        GetEndpointFromOrchestrationForm.endpoint TO F_EQ.IN2;
        F_EQ.OUT TO NoServiceAvailable.check;
        E_SR.Q TO SERVER_1.QI;
        Service1.arrowheadService TO RegisterService2.providedService;
        FieldsToArrowheadSystem.arrowheadSystem TO RegisterService2.provider;
        GET_STRUCT_VALUE1.OUT TO GetEndpointFromOrchestrationForm.orchestrationForm;
        FieldsToServiceRequestForm.serviceRequestForm TO RequestOrchestrationForm.serviceRequestForm;
        RequestOrchestrationForm.orchestrationResponse TO GET_STRUCT_VALUE1.IN_ARRAY;
      END_CONNECTIONS
      ADAPTER_CONNECTIONS
        RequestOrchestrationForm.requestOrchestration TO RequestOrchestrationHTTP.requestOrchestration;
      END_CONNECTIONS
    END_RESOURCE
    RESOURCE OrchestrationWithRules : EMB_RES
      FBS
        FieldsToArrowheadSystem : FieldsToArrowheadSystem(systemName := %systemName%, address := %testAddress%, port := %systemPort%);
        Service1 : FieldsToArrowheadService(serviceDefinition := %serviceDefinition%, interfaces := ["JSON", "XML"], serviceMetadata := %serviceMetadata%);
        F_EQ : F_EQ(IN1 := %emptyEndpoint%);
        NoServiceAvailable : TEST_CONDITION;
        SERVER_1 : SERVER_1(ID := http[/serviceTest/start]);
        E_SR : E_SR;
        SUBL_0 : SUBL_0(ID := %test7Ended%);
        PUBL_0 : PUBL_0(ID := %test8Ended%);
        F_EQ_1 : F_EQ(IN1 := %validEndpoint%);
        ServiceAvailable : TEST_CONDITION;
        E_SR_1 : E_SR;
        E_SWITCH : E_SWITCH;
        CLIENT_1_2 : CLIENT_1_2(QI := 1, ID := http[%authRuleEndpoint%; POST; application/json]], SD_1 := STRING#%authRuleData%);
        CLIENT_1_2_1 : CLIENT_1_2(QI := 1, ID := http[%orchStoreEndpoint%; POST; application/json]], SD_1 := STRING#%orchRuleData%);
        STRING2STRING : STRING2STRING;
      END_FBS
      SUBAPPS
        RegisterService2 : RegisterServicePartialHTTP(serviceURI := %serviceURI%, version := %serviceVersion%, udp := false, metadata := %metadata%, SRendpoint := %serviceRegistryAddress%);
        GetEndpointFromOrchestrationHTTPPFull : GetEndpointFromOrchestrationHTTPPFull(systemName := %systemName%, address := %testAddress%, port := %systemPort%, serviceDefinition := %serviceDefinition%, interfaces := ["JSON", "XML"], serviceMetadata := %serviceMetadata%, orchestratorEndpoint := %orchestratorAddress%, INDEX := 0);
      END_SUBAPPS
      SUBAPPLICATION Sequencer_1
        EVENT_INPUT
          Next;
        END_EVENT
        EVENT_OUTPUT
          E0;
          E1;
          E2;
          E3;
          E4;
          E5;
          E6;
          E7;
          E8;
          E9;
          E10;
          E11;
          E12;
          E13;
          E14;
          E15;
        END_EVENT
      END_SUBAPPLICATION
      EVENT_CONNECTIONS
        FieldsToArrowheadSystem.CNF TO Service1.REQ;
        F_EQ.CNF TO NoServiceAvailable.REQ;
        E_SR.EO TO SERVER_1.INIT;
        SUBL_0.IND TO FieldsToArrowheadSystem.REQ;
        RegisterService2.doneUnregister TO Sequencer_1.Next;
        RegisterService2.doneRegister TO Sequencer_1.Next;
        NoServiceAvailable.CNF TO Sequencer_1.Next;
        F_EQ_1.CNF TO ServiceAvailable.REQ;
        E_SWITCH.EO0 TO F_EQ.REQ;
        E_SWITCH.EO1 TO F_EQ_1.REQ;
        Sequencer_1.E2 TO RegisterService2.register;
        E_SR_1.EO TO Sequencer_1.Next;
        START.WARM TO SUBL_0.INIT;
        SERVER_1.INITO TO Sequencer_1.Next;
        CLIENT_1_2.INITO TO CLIENT_1_2.REQ;
        CLIENT_1_2.CNF TO CLIENT_1_2_1.INIT;
        CLIENT_1_2_1.INITO TO CLIENT_1_2_1.REQ;
        Sequencer_1.E0 TO CLIENT_1_2.INIT;
        SERVER_1.IND TO STRING2STRING.REQ;
        STRING2STRING.CNF TO SERVER_1.RSP;
        Sequencer_1.E3 TO E_SR_1.S;
        Sequencer_1.E5 TO E_SR.S;
        Sequencer_1.E7 TO RegisterService2.unregister;
        Sequencer_1.E8 TO E_SR_1.R;
        Sequencer_1.E10 TO E_SR.R;
        START.COLD TO SUBL_0.INIT;
        Service1.CNF TO Sequencer_1.Next;
        Sequencer_1.E11 TO GetEndpointFromOrchestrationHTTPPFull.REQ;
        Sequencer_1.E9 TO GetEndpointFromOrchestrationHTTPPFull.REQ;
        Sequencer_1.E6 TO GetEndpointFromOrchestrationHTTPPFull.REQ;
        Sequencer_1.E4 TO GetEndpointFromOrchestrationHTTPPFull.REQ;
        Sequencer_1.E1 TO GetEndpointFromOrchestrationHTTPPFull.REQ;
        GetEndpointFromOrchestrationHTTPPFull.CNF TO E_SWITCH.EI;
        CLIENT_1_2_1.CNF TO Sequencer_1.Next;
        ServiceAvailable.CNF TO Sequencer_1.Next;
        SUBL_0.INITO TO PUBL_0.INIT;
        Sequencer_1.E12 TO PUBL_0.REQ;
      END_CONNECTIONS
      DATA_CONNECTIONS
        F_EQ.OUT TO NoServiceAvailable.check;
        E_SR.Q TO SERVER_1.QI;
        Service1.arrowheadService TO RegisterService2.providedService;
        FieldsToArrowheadSystem.arrowheadSystem TO RegisterService2.provider;
        F_EQ_1.OUT TO ServiceAvailable.check;
        E_SR_1.Q TO E_SWITCH.G;
        SERVER_1.RD_1 TO STRING2STRING.IN;
        STRING2STRING.OUT TO SERVER_1.SD_1;
        GetEndpointFromOrchestrationHTTPPFull.endpoint TO F_EQ_1.IN2;
        GetEndpointFromOrchestrationHTTPPFull.endpoint TO F_EQ.IN2;
      END_CONNECTIONS
    END_RESOURCE
    RESOURCE PublishSubscribe : EMB_RES
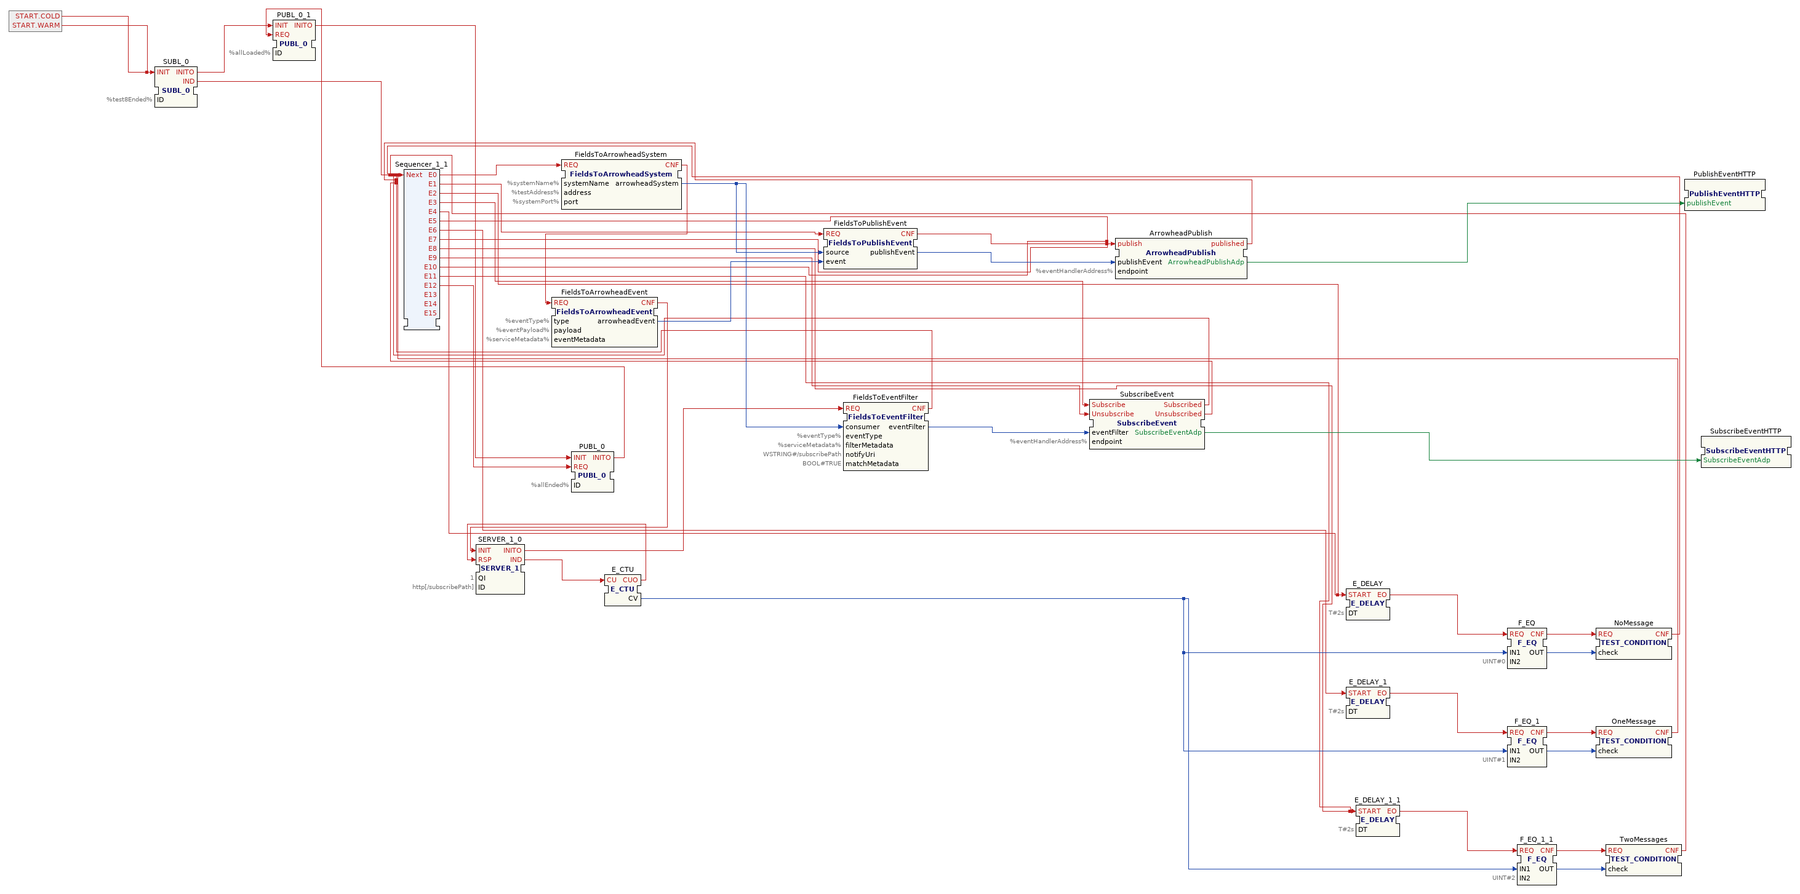
      FBS
        FieldsToArrowheadSystem : FieldsToArrowheadSystem(systemName := %systemName%, address := %testAddress%, port := %systemPort%);
        FieldsToPublishEvent : FieldsToPublishEvent;
        ArrowheadPublish : ArrowheadPublish(endpoint := %eventHandlerAddress%);
        FieldsToArrowheadEvent : FieldsToArrowheadEvent(type := %eventType%, payload := %eventPayload%, eventMetadata := %serviceMetadata%);
        SubscribeEvent : SubscribeEvent(endpoint := %eventHandlerAddress%);
        FieldsToEventFilter : FieldsToEventFilter(eventType := %eventType%, filterMetadata := %serviceMetadata%, notifyUri := WSTRING#/subscribePath, matchMetadata := BOOL#TRUE);
        E_CTU : E_CTU;
        F_EQ : F_EQ(IN2 := UINT#0);
        E_DELAY : E_DELAY(DT := T#2s);
        NoMessage : TEST_CONDITION;
        E_DELAY_1 : E_DELAY(DT := T#2s);
        F_EQ_1 : F_EQ(IN2 := UINT#1);
        OneMessage : TEST_CONDITION;
        E_DELAY_1_1 : E_DELAY(DT := T#2s);
        TwoMessages : TEST_CONDITION;
        F_EQ_1_1 : F_EQ(IN2 := UINT#2);
        SERVER_1_0 : SERVER_1(QI := 1, ID := http[/subscribePath]);
        PUBL_0_1 : PUBL_0(ID := %allLoaded%);
        SUBL_0 : SUBL_0(ID := %test8Ended%);
        PUBL_0 : PUBL_0(ID := %allEnded%);
        PublishEventHTTP : PublishEventHTTP;
        SubscribeEventHTTP : SubscribeEventHTTP;
      END_FBS
      SUBAPPLICATION Sequencer_1_1
        EVENT_INPUT
          Next;
        END_EVENT
        EVENT_OUTPUT
          E0;
          E1;
          E2;
          E3;
          E4;
          E5;
          E6;
          E7;
          E8;
          E9;
          E10;
          E11;
          E12;
          E13;
          E14;
          E15;
        END_EVENT
      END_SUBAPPLICATION
      EVENT_CONNECTIONS
        FieldsToPublishEvent.CNF TO ArrowheadPublish.publish;
        FieldsToArrowheadSystem.CNF TO FieldsToArrowheadEvent.REQ;
        E_DELAY.EO TO F_EQ.REQ;
        F_EQ.CNF TO NoMessage.REQ;
        E_DELAY_1.EO TO F_EQ_1.REQ;
        F_EQ_1.CNF TO OneMessage.REQ;
        E_DELAY_1_1.EO TO F_EQ_1_1.REQ;
        F_EQ_1_1.CNF TO TwoMessages.REQ;
        TwoMessages.CNF TO Sequencer_1_1.Next;
        OneMessage.CNF TO Sequencer_1_1.Next;
        NoMessage.CNF TO Sequencer_1_1.Next;
        FieldsToEventFilter.CNF TO Sequencer_1_1.Next;
        Sequencer_1_1.E0 TO FieldsToArrowheadSystem.REQ;
        Sequencer_1_1.E1 TO FieldsToPublishEvent.REQ;
        Sequencer_1_1.E2 TO E_DELAY.START;
        Sequencer_1_1.E3 TO SubscribeEvent.Subscribe;
        Sequencer_1_1.E4 TO E_DELAY.START;
        Sequencer_1_1.E5 TO ArrowheadPublish.publish;
        Sequencer_1_1.E6 TO E_DELAY_1.START;
        Sequencer_1_1.E7 TO ArrowheadPublish.publish;
        Sequencer_1_1.E8 TO E_DELAY_1_1.START;
        Sequencer_1_1.E9 TO SubscribeEvent.Unsubscribe;
        Sequencer_1_1.E10 TO ArrowheadPublish.publish;
        Sequencer_1_1.E11 TO E_DELAY_1_1.START;
        ArrowheadPublish.published TO Sequencer_1_1.Next;
        SubscribeEvent.Subscribed TO Sequencer_1_1.Next;
        FieldsToArrowheadEvent.CNF TO SERVER_1_0.INIT;
        E_CTU.CUO TO SERVER_1_0.RSP;
        SERVER_1_0.INITO TO FieldsToEventFilter.REQ;
        SERVER_1_0.IND TO E_CTU.CU;
        SubscribeEvent.Unsubscribed TO Sequencer_1_1.Next;
        SUBL_0.INITO TO PUBL_0_1.INIT;
        START.COLD TO SUBL_0.INIT;
        START.WARM TO SUBL_0.INIT;
        SUBL_0.IND TO Sequencer_1_1.Next;
        PUBL_0_1.INITO TO PUBL_0.INIT;
        PUBL_0.INITO TO PUBL_0_1.REQ;
        Sequencer_1_1.E12 TO PUBL_0.REQ;
      END_CONNECTIONS
      DATA_CONNECTIONS
        FieldsToArrowheadSystem.arrowheadSystem TO FieldsToPublishEvent.source;
        FieldsToPublishEvent.publishEvent TO ArrowheadPublish.publishEvent;
        FieldsToArrowheadEvent.arrowheadEvent TO FieldsToPublishEvent.event;
        FieldsToArrowheadSystem.arrowheadSystem TO FieldsToEventFilter.consumer;
        FieldsToEventFilter.eventFilter TO SubscribeEvent.eventFilter;
        E_CTU.CV TO F_EQ.IN1;
        F_EQ.OUT TO NoMessage.check;
        E_CTU.CV TO F_EQ_1.IN1;
        F_EQ_1.OUT TO OneMessage.check;
        F_EQ_1_1.OUT TO TwoMessages.check;
        E_CTU.CV TO F_EQ_1_1.IN1;
      END_CONNECTIONS
      ADAPTER_CONNECTIONS
        ArrowheadPublish.ArrowheadPublishAdp TO PublishEventHTTP.publishEvent;
        SubscribeEvent.SubscribeEventAdp TO SubscribeEventHTTP.SubscribeEventAdp;
      END_CONNECTIONS
    END_RESOURCE
  END_DEVICE
  DEVICE OpcUaTest : FORTE_PC(MGR_ID := %opcuaTestAddress%)
    {SET_ATTRIBUTE(Profile, HOLOBLOC)} (* device profile *)
    RESOURCE cleanAll : EMB_RES
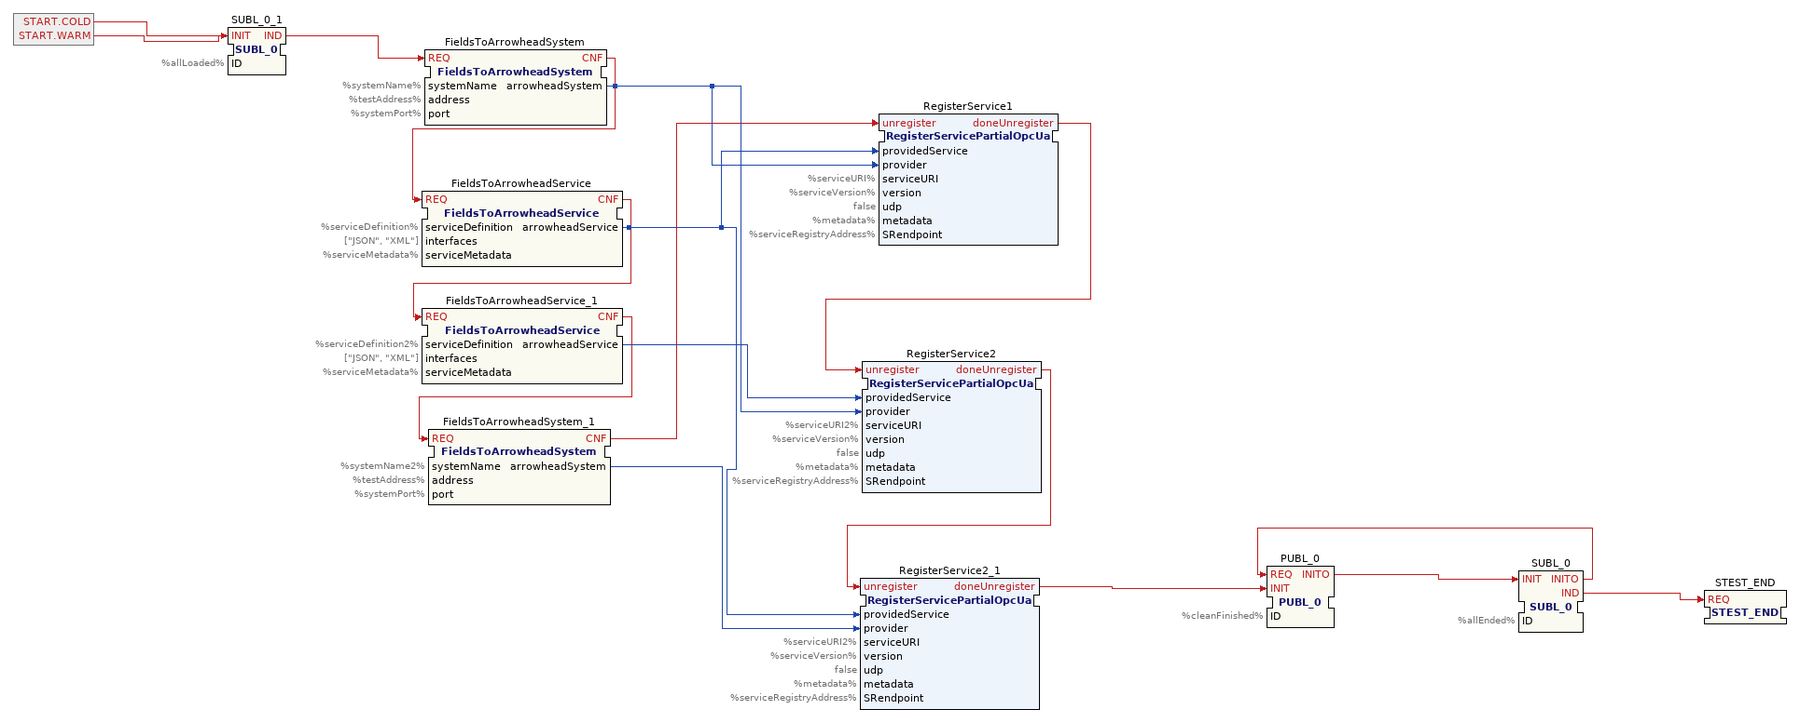
      FBS
        PUBL_0 : PUBL_0(ID := %cleanFinished%);
        FieldsToArrowheadSystem : FieldsToArrowheadSystem(systemName := %systemName%, address := %testAddress%, port := %systemPort%);
        FieldsToArrowheadService : FieldsToArrowheadService(serviceDefinition := %serviceDefinition%, interfaces := ["JSON", "XML"], serviceMetadata := %serviceMetadata%);
        FieldsToArrowheadService_1 : FieldsToArrowheadService(serviceDefinition := %serviceDefinition2%, interfaces := ["JSON", "XML"], serviceMetadata := %serviceMetadata%);
        FieldsToArrowheadSystem_1 : FieldsToArrowheadSystem(systemName := %systemName2%, address := %testAddress%, port := %systemPort%);
        SUBL_0 : SUBL_0(ID := %allEnded%);
        STEST_END : STEST_END;
        SUBL_0_1 : SUBL_0(ID := %allLoaded%);
      END_FBS
      SUBAPPS
        RegisterService1 : RegisterServicePartialOpcUa(serviceURI := %serviceURI%, version := %serviceVersion%, udp := false, metadata := %metadata%, SRendpoint := %serviceRegistryAddress%);
        RegisterService2_1 : RegisterServicePartialOpcUa(serviceURI := %serviceURI2%, version := %serviceVersion%, udp := false, metadata := %metadata%, SRendpoint := %serviceRegistryAddress%);
        RegisterService2 : RegisterServicePartialOpcUa(serviceURI := %serviceURI2%, version := %serviceVersion%, udp := false, metadata := %metadata%, SRendpoint := %serviceRegistryAddress%);
      END_SUBAPPS
      EVENT_CONNECTIONS
        FieldsToArrowheadSystem.CNF TO FieldsToArrowheadService.REQ;
        FieldsToArrowheadService.CNF TO FieldsToArrowheadService_1.REQ;
        FieldsToArrowheadService_1.CNF TO FieldsToArrowheadSystem_1.REQ;
        PUBL_0.INITO TO SUBL_0.INIT;
        SUBL_0.INITO TO PUBL_0.REQ;
        SUBL_0.IND TO STEST_END.REQ;
        START.COLD TO SUBL_0_1.INIT;
        START.WARM TO SUBL_0_1.INIT;
        FieldsToArrowheadSystem_1.CNF TO RegisterService1.unregister;
        RegisterService2_1.doneUnregister TO PUBL_0.INIT;
        RegisterService1.doneUnregister TO RegisterService2.unregister;
        RegisterService2.doneUnregister TO RegisterService2_1.unregister;
        SUBL_0_1.IND TO FieldsToArrowheadSystem.REQ;
      END_CONNECTIONS
      DATA_CONNECTIONS
        FieldsToArrowheadService.arrowheadService TO RegisterService1.providedService;
        FieldsToArrowheadSystem.arrowheadSystem TO RegisterService1.provider;
        FieldsToArrowheadService.arrowheadService TO RegisterService2_1.providedService;
        FieldsToArrowheadSystem_1.arrowheadSystem TO RegisterService2_1.provider;
        FieldsToArrowheadService_1.arrowheadService TO RegisterService2.providedService;
        FieldsToArrowheadSystem.arrowheadSystem TO RegisterService2.provider;
      END_CONNECTIONS
    END_RESOURCE
    RESOURCE RegisterUnregister : EMB_RES
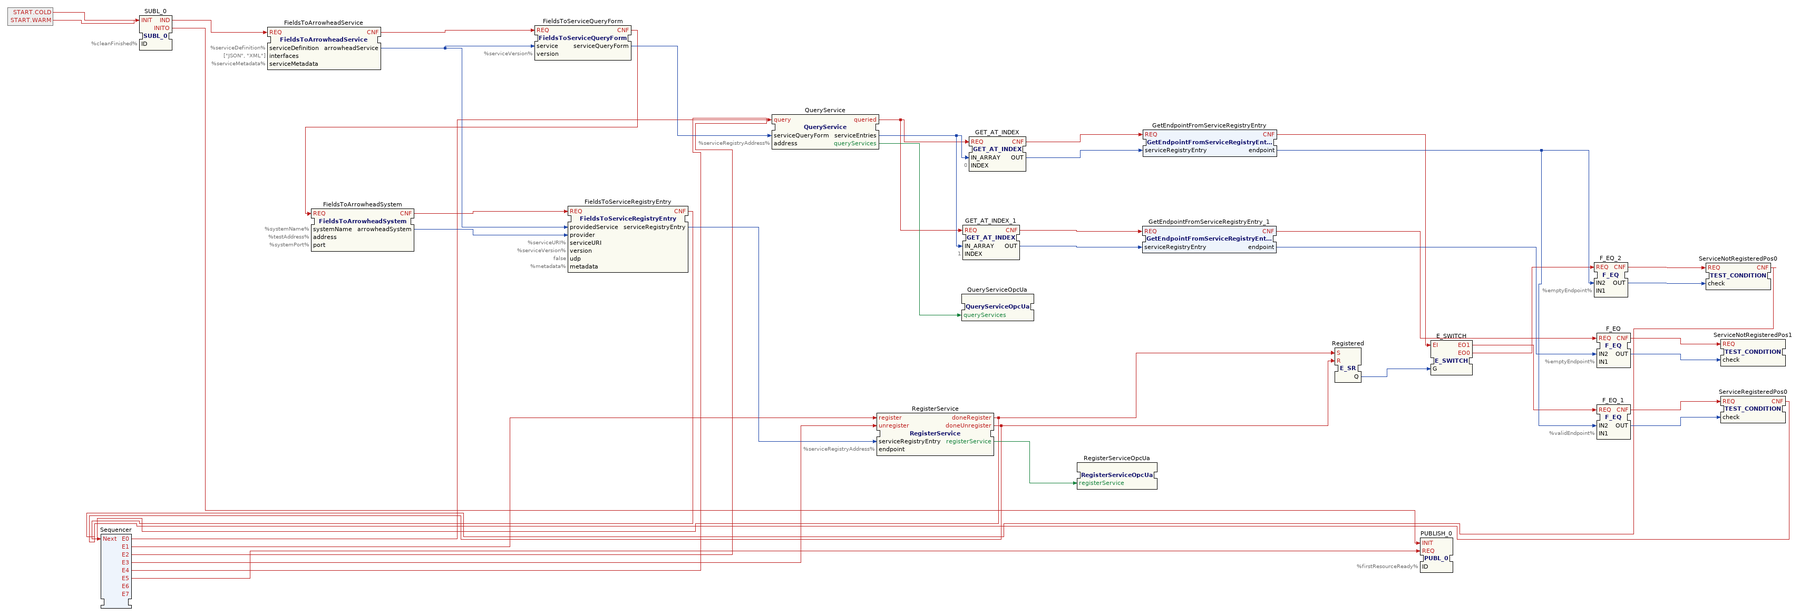
      FBS
        QueryService : QueryService(address := %serviceRegistryAddress%);
        GET_AT_INDEX : GET_AT_INDEX(INDEX := 0);
        F_EQ : F_EQ(IN1 := %emptyEndpoint%);
        ServiceNotRegisteredPos1 : TEST_CONDITION;
        FieldsToArrowheadService : FieldsToArrowheadService(serviceDefinition := %serviceDefinition%, interfaces := ["JSON", "XML"], serviceMetadata := %serviceMetadata%);
        FieldsToServiceQueryForm : FieldsToServiceQueryForm(version := %serviceVersion%);
        Registered : E_SR;
        E_SWITCH : E_SWITCH;
        F_EQ_1 : F_EQ(IN1 := %validEndpoint%);
        ServiceRegisteredPos0 : TEST_CONDITION;
        FieldsToArrowheadSystem : FieldsToArrowheadSystem(systemName := %systemName%, address := %testAddress%, port := %systemPort%);
        FieldsToServiceRegistryEntry : FieldsToServiceRegistryEntry(serviceURI := %serviceURI%, version := %serviceVersion%, udp := false, metadata := %metadata%);
        RegisterService : RegisterService(endpoint := %serviceRegistryAddress%);
        ServiceNotRegisteredPos0 : TEST_CONDITION;
        GET_AT_INDEX_1 : GET_AT_INDEX(INDEX := 1);
        F_EQ_2 : F_EQ(IN1 := %emptyEndpoint%);
        PUBLISH_0 : PUBL_0(ID := %firstResourceReady%);
        SUBL_0 : SUBL_0(ID := %cleanFinished%);
        RegisterServiceOpcUa : RegisterServiceOpcUa;
        QueryServiceOpcUa : QueryServiceOpcUa;
      END_FBS
      SUBAPPS
        GetEndpointFromServiceRegistryEntry : GetEndpointFromServiceRegistryEntry;
        GetEndpointFromServiceRegistryEntry_1 : GetEndpointFromServiceRegistryEntry;
      END_SUBAPPS
      SUBAPPLICATION Sequencer
        EVENT_INPUT
          Next;
        END_EVENT
        EVENT_OUTPUT
          E0;
          E1;
          E2;
          E3;
          E4;
          E5;
          E6;
          E7;
        END_EVENT
      END_SUBAPPLICATION
      EVENT_CONNECTIONS
        QueryService.queried TO GET_AT_INDEX.REQ;
        F_EQ.CNF TO ServiceNotRegisteredPos1.REQ;
        GET_AT_INDEX.CNF TO GetEndpointFromServiceRegistryEntry.REQ;
        FieldsToArrowheadService.CNF TO FieldsToServiceQueryForm.REQ;
        GetEndpointFromServiceRegistryEntry.CNF TO E_SWITCH.EI;
        E_SWITCH.EO1 TO F_EQ_1.REQ;
        F_EQ_1.CNF TO ServiceRegisteredPos0.REQ;
        ServiceRegisteredPos0.CNF TO Sequencer.Next;
        Sequencer.E0 TO QueryService.query;
        Sequencer.E2 TO QueryService.query;
        Sequencer.E4 TO QueryService.query;
        FieldsToServiceQueryForm.CNF TO FieldsToArrowheadSystem.REQ;
        FieldsToArrowheadSystem.CNF TO FieldsToServiceRegistryEntry.REQ;
        FieldsToServiceRegistryEntry.CNF TO Sequencer.Next;
        Sequencer.E1 TO RegisterService.register;
        Sequencer.E3 TO RegisterService.unregister;
        RegisterService.doneRegister TO Sequencer.Next;
        RegisterService.doneRegister TO Registered.S;
        RegisterService.doneUnregister TO Sequencer.Next;
        RegisterService.doneUnregister TO Registered.R;
        GetEndpointFromServiceRegistryEntry_1.CNF TO F_EQ.REQ;
        ServiceNotRegisteredPos0.CNF TO Sequencer.Next;
        QueryService.queried TO GET_AT_INDEX_1.REQ;
        GET_AT_INDEX_1.CNF TO GetEndpointFromServiceRegistryEntry_1.REQ;
        E_SWITCH.EO0 TO F_EQ_2.REQ;
        F_EQ_2.CNF TO ServiceNotRegisteredPos0.REQ;
        SUBL_0.IND TO FieldsToArrowheadService.REQ;
        START.COLD TO SUBL_0.INIT;
        START.WARM TO SUBL_0.INIT;
        SUBL_0.INITO TO PUBLISH_0.INIT;
        Sequencer.E5 TO PUBLISH_0.REQ;
      END_CONNECTIONS
      DATA_CONNECTIONS
        QueryService.serviceEntries TO GET_AT_INDEX.IN_ARRAY;
        F_EQ.OUT TO ServiceNotRegisteredPos1.check;
        GET_AT_INDEX.OUT TO GetEndpointFromServiceRegistryEntry.serviceRegistryEntry;
        FieldsToArrowheadService.arrowheadService TO FieldsToServiceQueryForm.service;
        FieldsToServiceQueryForm.serviceQueryForm TO QueryService.serviceQueryForm;
        Registered.Q TO E_SWITCH.G;
        GetEndpointFromServiceRegistryEntry.endpoint TO F_EQ_1.IN2;
        F_EQ_1.OUT TO ServiceRegisteredPos0.check;
        FieldsToArrowheadService.arrowheadService TO FieldsToServiceRegistryEntry.providedService;
        FieldsToArrowheadSystem.arrowheadSystem TO FieldsToServiceRegistryEntry.provider;
        FieldsToServiceRegistryEntry.serviceRegistryEntry TO RegisterService.serviceRegistryEntry;
        GetEndpointFromServiceRegistryEntry_1.endpoint TO F_EQ.IN2;
        QueryService.serviceEntries TO GET_AT_INDEX_1.IN_ARRAY;
        GET_AT_INDEX_1.OUT TO GetEndpointFromServiceRegistryEntry_1.serviceRegistryEntry;
        GetEndpointFromServiceRegistryEntry.endpoint TO F_EQ_2.IN2;
        F_EQ_2.OUT TO ServiceNotRegisteredPos0.check;
      END_CONNECTIONS
      ADAPTER_CONNECTIONS
        RegisterService.registerService TO RegisterServiceOpcUa.registerService;
        QueryService.queryServices TO QueryServiceOpcUa.queryServices;
      END_CONNECTIONS
    END_RESOURCE
    RESOURCE DoubleRegister : EMB_RES
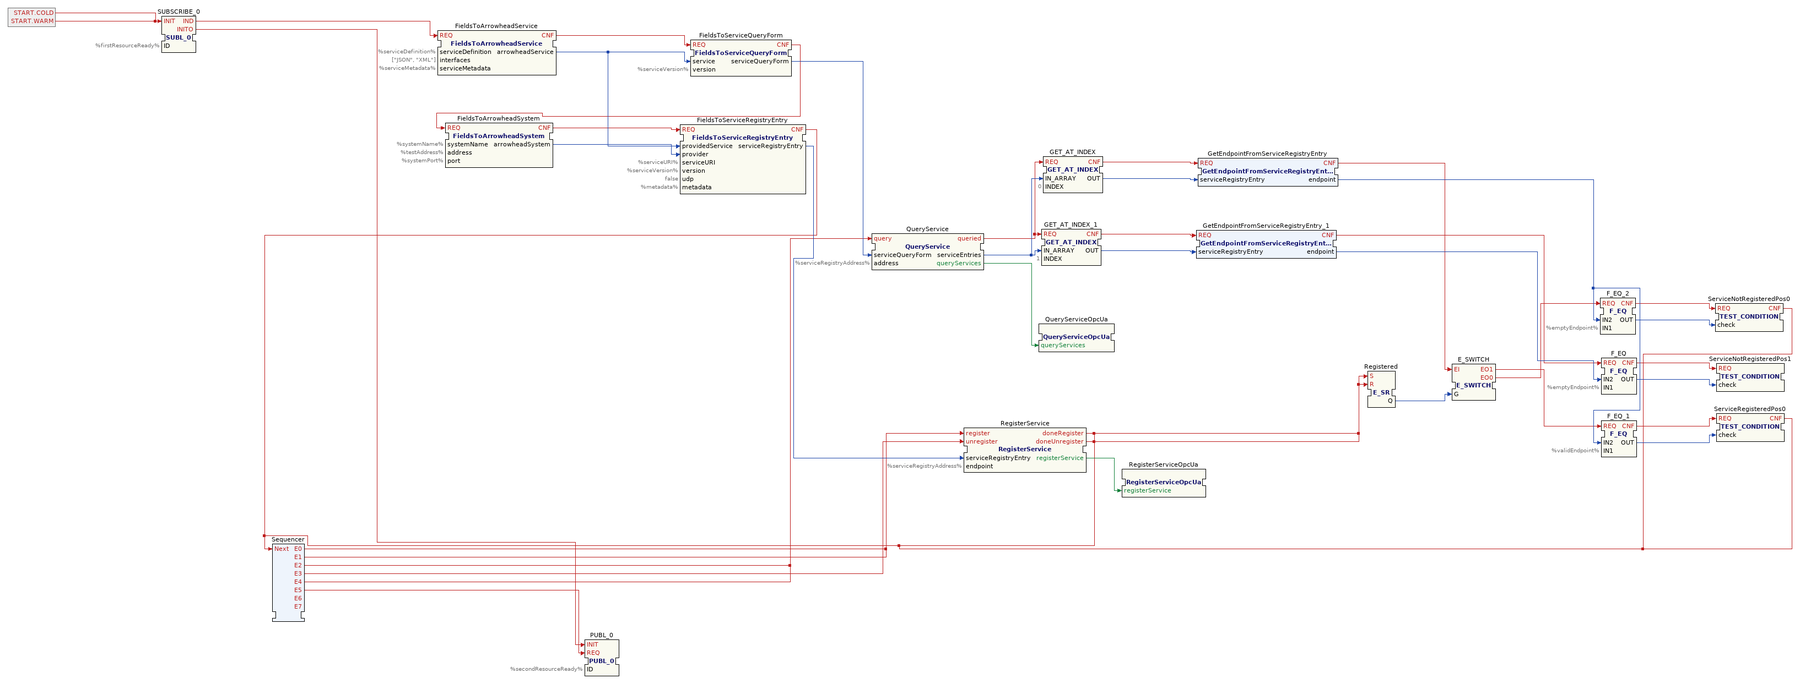
      FBS
        QueryService : QueryService(address := %serviceRegistryAddress%);
        GET_AT_INDEX : GET_AT_INDEX(INDEX := 0);
        F_EQ : F_EQ(IN1 := %emptyEndpoint%);
        ServiceNotRegisteredPos1 : TEST_CONDITION;
        FieldsToArrowheadService : FieldsToArrowheadService(serviceDefinition := %serviceDefinition%, interfaces := ["JSON", "XML"], serviceMetadata := %serviceMetadata%);
        FieldsToServiceQueryForm : FieldsToServiceQueryForm(version := %serviceVersion%);
        Registered : E_SR;
        E_SWITCH : E_SWITCH;
        F_EQ_1 : F_EQ(IN1 := %validEndpoint%);
        ServiceRegisteredPos0 : TEST_CONDITION;
        FieldsToArrowheadSystem : FieldsToArrowheadSystem(systemName := %systemName%, address := %testAddress%, port := %systemPort%);
        FieldsToServiceRegistryEntry : FieldsToServiceRegistryEntry(serviceURI := %serviceURI%, version := %serviceVersion%, udp := false, metadata := %metadata%);
        RegisterService : RegisterService(endpoint := %serviceRegistryAddress%);
        GET_AT_INDEX_1 : GET_AT_INDEX(INDEX := 1);
        F_EQ_2 : F_EQ(IN1 := %emptyEndpoint%);
        ServiceNotRegisteredPos0 : TEST_CONDITION;
        SUBSCRIBE_0 : SUBL_0(ID := %firstResourceReady%);
        PUBL_0 : PUBL_0(ID := %secondResourceReady%);
        RegisterServiceOpcUa : RegisterServiceOpcUa;
        QueryServiceOpcUa : QueryServiceOpcUa;
      END_FBS
      SUBAPPS
        GetEndpointFromServiceRegistryEntry : GetEndpointFromServiceRegistryEntry;
        GetEndpointFromServiceRegistryEntry_1 : GetEndpointFromServiceRegistryEntry;
      END_SUBAPPS
      SUBAPPLICATION Sequencer
        EVENT_INPUT
          Next;
        END_EVENT
        EVENT_OUTPUT
          E0;
          E1;
          E2;
          E3;
          E4;
          E5;
          E6;
          E7;
        END_EVENT
      END_SUBAPPLICATION
      EVENT_CONNECTIONS
        QueryService.queried TO GET_AT_INDEX.REQ;
        F_EQ.CNF TO ServiceNotRegisteredPos1.REQ;
        GET_AT_INDEX.CNF TO GetEndpointFromServiceRegistryEntry.REQ;
        FieldsToArrowheadService.CNF TO FieldsToServiceQueryForm.REQ;
        GetEndpointFromServiceRegistryEntry.CNF TO E_SWITCH.EI;
        E_SWITCH.EO1 TO F_EQ_1.REQ;
        F_EQ_1.CNF TO ServiceRegisteredPos0.REQ;
        ServiceRegisteredPos0.CNF TO Sequencer.Next;
        Sequencer.E2 TO QueryService.query;
        Sequencer.E4 TO QueryService.query;
        FieldsToServiceQueryForm.CNF TO FieldsToArrowheadSystem.REQ;
        FieldsToArrowheadSystem.CNF TO FieldsToServiceRegistryEntry.REQ;
        FieldsToServiceRegistryEntry.CNF TO Sequencer.Next;
        Sequencer.E0 TO RegisterService.register;
        Sequencer.E1 TO RegisterService.register;
        Sequencer.E3 TO RegisterService.unregister;
        RegisterService.doneRegister TO Registered.S;
        RegisterService.doneRegister TO Sequencer.Next;
        RegisterService.doneUnregister TO Registered.R;
        RegisterService.doneUnregister TO Sequencer.Next;
        GetEndpointFromServiceRegistryEntry_1.CNF TO F_EQ.REQ;
        QueryService.queried TO GET_AT_INDEX_1.REQ;
        GET_AT_INDEX_1.CNF TO GetEndpointFromServiceRegistryEntry_1.REQ;
        E_SWITCH.EO0 TO F_EQ_2.REQ;
        F_EQ_2.CNF TO ServiceNotRegisteredPos0.REQ;
        ServiceNotRegisteredPos0.CNF TO Sequencer.Next;
        SUBSCRIBE_0.IND TO FieldsToArrowheadService.REQ;
        SUBSCRIBE_0.INITO TO PUBL_0.INIT;
        Sequencer.E5 TO PUBL_0.REQ;
        START.COLD TO SUBSCRIBE_0.INIT;
        START.WARM TO SUBSCRIBE_0.INIT;
      END_CONNECTIONS
      DATA_CONNECTIONS
        QueryService.serviceEntries TO GET_AT_INDEX.IN_ARRAY;
        F_EQ.OUT TO ServiceNotRegisteredPos1.check;
        GET_AT_INDEX.OUT TO GetEndpointFromServiceRegistryEntry.serviceRegistryEntry;
        FieldsToArrowheadService.arrowheadService TO FieldsToServiceQueryForm.service;
        FieldsToServiceQueryForm.serviceQueryForm TO QueryService.serviceQueryForm;
        Registered.Q TO E_SWITCH.G;
        GetEndpointFromServiceRegistryEntry.endpoint TO F_EQ_1.IN2;
        F_EQ_1.OUT TO ServiceRegisteredPos0.check;
        FieldsToArrowheadService.arrowheadService TO FieldsToServiceRegistryEntry.providedService;
        FieldsToArrowheadSystem.arrowheadSystem TO FieldsToServiceRegistryEntry.provider;
        FieldsToServiceRegistryEntry.serviceRegistryEntry TO RegisterService.serviceRegistryEntry;
        GetEndpointFromServiceRegistryEntry_1.endpoint TO F_EQ.IN2;
        QueryService.serviceEntries TO GET_AT_INDEX_1.IN_ARRAY;
        GET_AT_INDEX_1.OUT TO GetEndpointFromServiceRegistryEntry_1.serviceRegistryEntry;
        GetEndpointFromServiceRegistryEntry.endpoint TO F_EQ_2.IN2;
        F_EQ_2.OUT TO ServiceNotRegisteredPos0.check;
      END_CONNECTIONS
      ADAPTER_CONNECTIONS
        RegisterService.registerService TO RegisterServiceOpcUa.registerService;
        QueryService.queryServices TO QueryServiceOpcUa.queryServices;
      END_CONNECTIONS
    END_RESOURCE
    RESOURCE RegisterMoreServices : EMB_RES
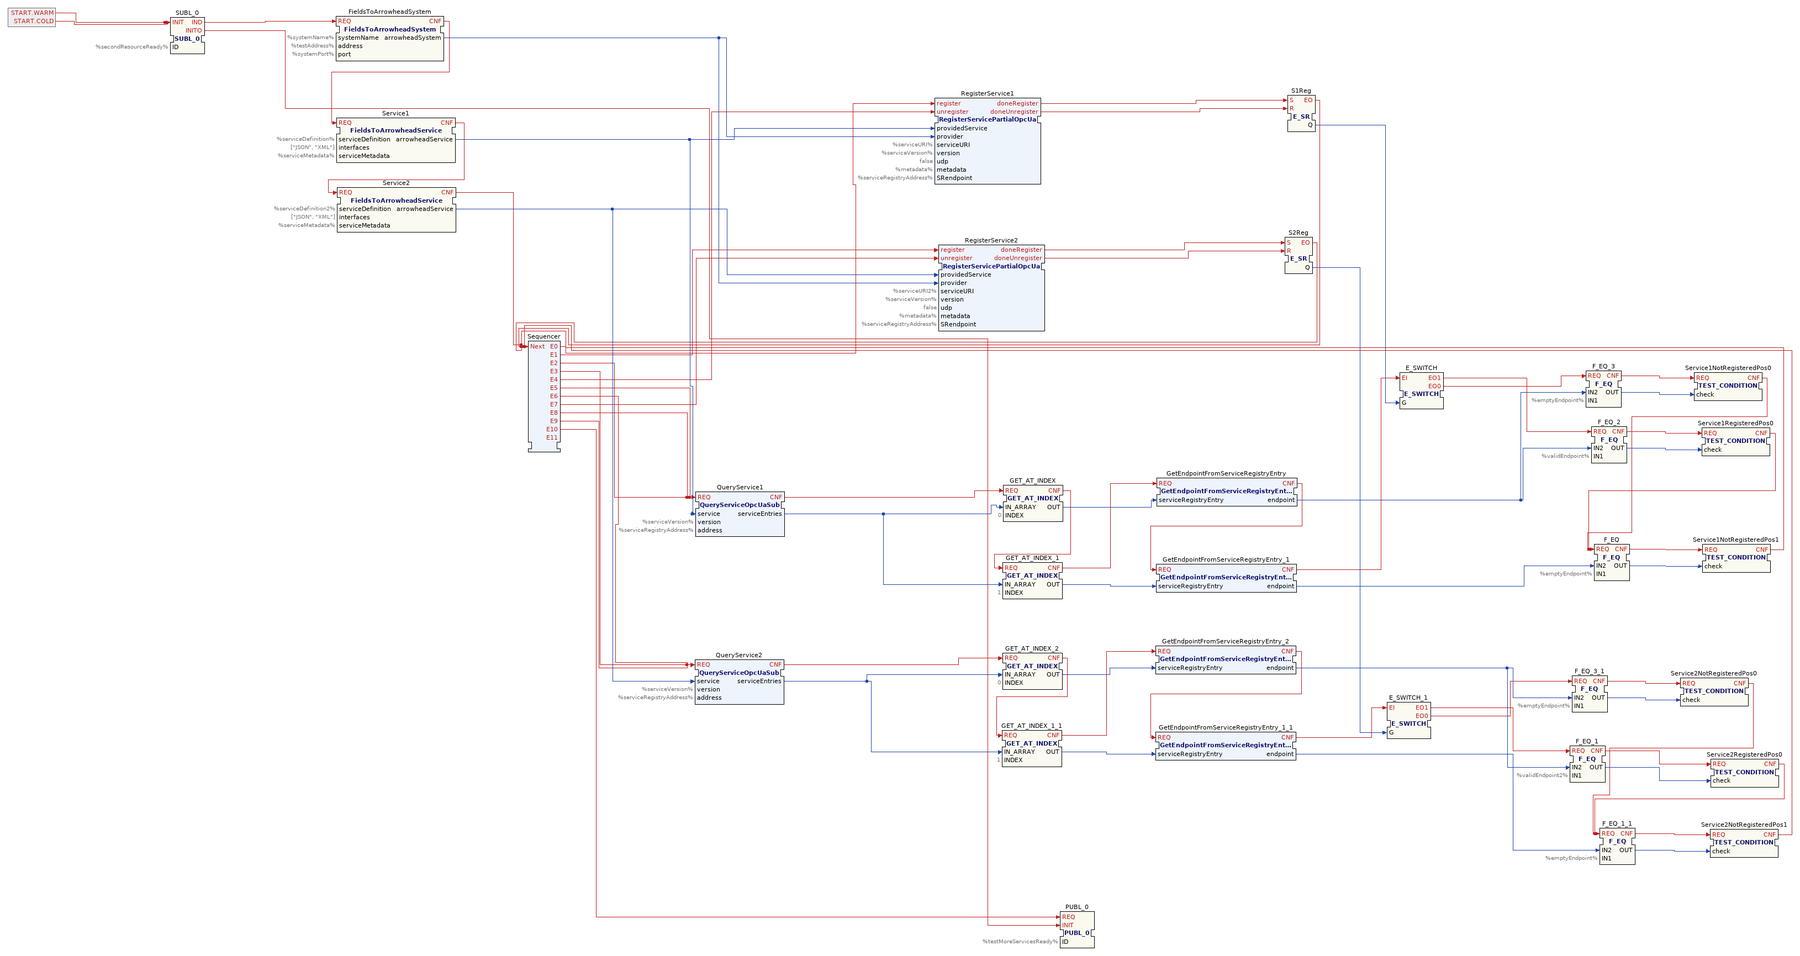
      FBS
        GET_AT_INDEX_1 : GET_AT_INDEX(INDEX := 1);
        F_EQ : F_EQ(IN1 := %emptyEndpoint%);
        FieldsToArrowheadSystem : FieldsToArrowheadSystem(systemName := %systemName%, address := %testAddress%, port := %systemPort%);
        F_EQ_2 : F_EQ(IN1 := %validEndpoint%);
        GET_AT_INDEX : GET_AT_INDEX(INDEX := 0);
        S1Reg : E_SR;
        Service2RegisteredPos0 : TEST_CONDITION;
        E_SWITCH : E_SWITCH;
        F_EQ_1 : F_EQ(IN1 := %validEndpoint2%);
        Service1RegisteredPos0 : TEST_CONDITION;
        Service1NotRegisteredPos1 : TEST_CONDITION;
        Service2NotRegisteredPos1 : TEST_CONDITION;
        F_EQ_1_1 : F_EQ(IN1 := %emptyEndpoint%);
        S2Reg : E_SR;
        E_SWITCH_1 : E_SWITCH;
        GET_AT_INDEX_1_1 : GET_AT_INDEX(INDEX := 1);
        GET_AT_INDEX_2 : GET_AT_INDEX(INDEX := 0);
        SUBL_0 : SUBL_0(ID := %secondResourceReady%);
        Service1NotRegisteredPos0 : TEST_CONDITION;
        F_EQ_3 : F_EQ(IN1 := %emptyEndpoint%);
        F_EQ_3_1 : F_EQ(IN1 := %emptyEndpoint%);
        Service2NotRegisteredPos0 : TEST_CONDITION;
        Service1 : FieldsToArrowheadService(serviceDefinition := %serviceDefinition%, interfaces := ["JSON", "XML"], serviceMetadata := %serviceMetadata%);
        Service2 : FieldsToArrowheadService(serviceDefinition := %serviceDefinition2%, interfaces := ["JSON", "XML"], serviceMetadata := %serviceMetadata%);
        PUBL_0 : PUBL_0(ID := %testMoreServicesReady%);
      END_FBS
      SUBAPPS
        GetEndpointFromServiceRegistryEntry_1 : GetEndpointFromServiceRegistryEntry;
        GetEndpointFromServiceRegistryEntry : GetEndpointFromServiceRegistryEntry;
        GetEndpointFromServiceRegistryEntry_1_1 : GetEndpointFromServiceRegistryEntry;
        GetEndpointFromServiceRegistryEntry_2 : GetEndpointFromServiceRegistryEntry;
        RegisterService2 : RegisterServicePartialOpcUa(serviceURI := %serviceURI2%, version := %serviceVersion%, udp := false, metadata := %metadata%, SRendpoint := %serviceRegistryAddress%);
        RegisterService1 : RegisterServicePartialOpcUa(serviceURI := %serviceURI%, version := %serviceVersion%, udp := false, metadata := %metadata%, SRendpoint := %serviceRegistryAddress%);
        QueryService2 : QueryServiceOpcUaSub(version := %serviceVersion%, address := %serviceRegistryAddress%);
        QueryService1 : QueryServiceOpcUaSub(version := %serviceVersion%, address := %serviceRegistryAddress%);
      END_SUBAPPS
      SUBAPPLICATION Sequencer
        EVENT_INPUT
          Next;
        END_EVENT
        EVENT_OUTPUT
          E0;
          E1;
          E2;
          E3;
          E4;
          E5;
          E6;
          E7;
          E8;
          E9;
          E10;
          E11;
        END_EVENT
      END_SUBAPPLICATION
      EVENT_CONNECTIONS
        GET_AT_INDEX_1.CNF TO GetEndpointFromServiceRegistryEntry.REQ;
        GetEndpointFromServiceRegistryEntry.CNF TO GetEndpointFromServiceRegistryEntry_1.REQ;
        GET_AT_INDEX.CNF TO GET_AT_INDEX_1.REQ;
        GetEndpointFromServiceRegistryEntry_1.CNF TO E_SWITCH.EI;
        E_SWITCH.EO1 TO F_EQ_2.REQ;
        F_EQ_1.CNF TO Service2RegisteredPos0.REQ;
        F_EQ_2.CNF TO Service1RegisteredPos0.REQ;
        Service1RegisteredPos0.CNF TO F_EQ.REQ;
        F_EQ.CNF TO Service1NotRegisteredPos1.REQ;
        Service1NotRegisteredPos1.CNF TO Sequencer.Next;
        S1Reg.EO TO Sequencer.Next;
        Service2NotRegisteredPos1.CNF TO Sequencer.Next;
        Service2RegisteredPos0.CNF TO F_EQ_1_1.REQ;
        F_EQ_1_1.CNF TO Service2NotRegisteredPos1.REQ;
        S2Reg.EO TO Sequencer.Next;
        E_SWITCH_1.EO1 TO F_EQ_1.REQ;
        GetEndpointFromServiceRegistryEntry_1_1.CNF TO E_SWITCH_1.EI;
        GET_AT_INDEX_1_1.CNF TO GetEndpointFromServiceRegistryEntry_2.REQ;
        GetEndpointFromServiceRegistryEntry_2.CNF TO GetEndpointFromServiceRegistryEntry_1_1.REQ;
        GET_AT_INDEX_2.CNF TO GET_AT_INDEX_1_1.REQ;
        SUBL_0.IND TO FieldsToArrowheadSystem.REQ;
        Service1NotRegisteredPos0.CNF TO F_EQ.REQ;
        E_SWITCH.EO0 TO F_EQ_3.REQ;
        F_EQ_3.CNF TO Service1NotRegisteredPos0.REQ;
        E_SWITCH_1.EO0 TO F_EQ_3_1.REQ;
        F_EQ_3_1.CNF TO Service2NotRegisteredPos0.REQ;
        Service2NotRegisteredPos0.CNF TO F_EQ_1_1.REQ;
        FieldsToArrowheadSystem.CNF TO Service1.REQ;
        Service1.CNF TO Service2.REQ;
        Service2.CNF TO Sequencer.Next;
        START.WARM TO SUBL_0.INIT;
        START.COLD TO SUBL_0.INIT;
        Sequencer.E1 TO RegisterService2.register;
        Sequencer.E7 TO RegisterService2.unregister;
        RegisterService2.doneRegister TO S2Reg.S;
        RegisterService2.doneUnregister TO S2Reg.R;
        Sequencer.E0 TO RegisterService1.register;
        Sequencer.E4 TO RegisterService1.unregister;
        RegisterService1.doneRegister TO S1Reg.S;
        RegisterService1.doneUnregister TO S1Reg.R;
        Sequencer.E3 TO QueryService2.REQ;
        Sequencer.E6 TO QueryService2.REQ;
        Sequencer.E9 TO QueryService2.REQ;
        QueryService2.CNF TO GET_AT_INDEX_2.REQ;
        Sequencer.E2 TO QueryService1.REQ;
        Sequencer.E5 TO QueryService1.REQ;
        Sequencer.E8 TO QueryService1.REQ;
        QueryService1.CNF TO GET_AT_INDEX.REQ;
        Sequencer.E10 TO PUBL_0.REQ;
        SUBL_0.INITO TO PUBL_0.INIT;
      END_CONNECTIONS
      DATA_CONNECTIONS
        GET_AT_INDEX_1.OUT TO GetEndpointFromServiceRegistryEntry_1.serviceRegistryEntry;
        GetEndpointFromServiceRegistryEntry_1.endpoint TO F_EQ.IN2;
        GetEndpointFromServiceRegistryEntry.endpoint TO F_EQ_2.IN2;
        GET_AT_INDEX.OUT TO GetEndpointFromServiceRegistryEntry.serviceRegistryEntry;
        S1Reg.Q TO E_SWITCH.G;
        F_EQ_1.OUT TO Service2RegisteredPos0.check;
        F_EQ_2.OUT TO Service1RegisteredPos0.check;
        F_EQ.OUT TO Service1NotRegisteredPos1.check;
        F_EQ_1_1.OUT TO Service2NotRegisteredPos1.check;
        S2Reg.Q TO E_SWITCH_1.G;
        GET_AT_INDEX_1_1.OUT TO GetEndpointFromServiceRegistryEntry_1_1.serviceRegistryEntry;
        GetEndpointFromServiceRegistryEntry_1_1.endpoint TO F_EQ_1_1.IN2;
        GetEndpointFromServiceRegistryEntry_2.endpoint TO F_EQ_1.IN2;
        GET_AT_INDEX_2.OUT TO GetEndpointFromServiceRegistryEntry_2.serviceRegistryEntry;
        GetEndpointFromServiceRegistryEntry.endpoint TO F_EQ_3.IN2;
        F_EQ_3.OUT TO Service1NotRegisteredPos0.check;
        GetEndpointFromServiceRegistryEntry_2.endpoint TO F_EQ_3_1.IN2;
        F_EQ_3_1.OUT TO Service2NotRegisteredPos0.check;
        Service2.arrowheadService TO RegisterService2.providedService;
        FieldsToArrowheadSystem.arrowheadSystem TO RegisterService2.provider;
        Service1.arrowheadService TO RegisterService1.providedService;
        FieldsToArrowheadSystem.arrowheadSystem TO RegisterService1.provider;
        Service2.arrowheadService TO QueryService2.service;
        QueryService2.serviceEntries TO GET_AT_INDEX_2.IN_ARRAY;
        QueryService2.serviceEntries TO GET_AT_INDEX_1_1.IN_ARRAY;
        Service1.arrowheadService TO QueryService1.service;
        QueryService1.serviceEntries TO GET_AT_INDEX.IN_ARRAY;
        QueryService1.serviceEntries TO GET_AT_INDEX_1.IN_ARRAY;
      END_CONNECTIONS
    END_RESOURCE
    RESOURCE SameServiceTwice : EMB_RES
      FBS
        SUBL_0 : SUBL_0(ID := %testMoreServicesReady%);
        Service1 : FieldsToArrowheadService(serviceDefinition := %serviceDefinition%, interfaces := ["JSON", "XML"], serviceMetadata := %serviceMetadata%);
        FieldsToArrowheadSystem : FieldsToArrowheadSystem(systemName := %systemName%, address := %testAddress%, port := %systemPort%);
        GET_AT_INDEX_1 : GET_AT_INDEX(INDEX := 1);
        GET_AT_INDEX : GET_AT_INDEX(INDEX := 0);
        Service1RegisteredPos0 : TEST_CONDITION;
        F_EQ_2 : F_EQ(IN1 := %validEndpoint%);
        BothServicesRegistered : TEST_CONDITION;
        F_EQ_3 : F_EQ(IN1 := %validEndpoint2%);
        F_EQ : F_EQ(IN1 := %validEndpoint%);
        F_EQ_2_1 : F_EQ(IN1 := %validEndpoint2%);
        F_EQ_3_1 : F_EQ(IN1 := %validEndpoint%);
        Service2RegisteredPos0 : TEST_CONDITION;
        F_EQ_1 : F_EQ(IN1 := %validEndpoint2%);
        BothServicesNotRegistered : TEST_CONDITION;
        F_EQ_1_1 : F_EQ(IN1 := %emptyEndpoint%);
        F_EQ_1_1_1 : F_EQ(IN1 := %emptyEndpoint%);
        Service2NotRegisteredPos1 : TEST_CONDITION;
        F_EQ_4 : F_EQ(IN1 := %emptyEndpoint%);
        F_EQ_4_1 : F_EQ(IN1 := %emptyEndpoint%);
        Service1NotRegisteredPos1 : TEST_CONDITION;
        F_AND : F_AND;
        E_MERGE : E_MERGE;
        E_MERGE_1 : E_MERGE;
        F_AND_1 : F_AND;
        F_OR : F_OR;
        F_AND_1_1 : F_AND;
        BOOL2BOOL : BOOL2BOOL;
        BOOL2BOOL_1 : BOOL2BOOL;
        FieldsToArrowheadSystem_1 : FieldsToArrowheadSystem(systemName := %systemName2%, address := %testAddress%, port := %systemPort%);
        PUBL_0 : PUBL_0(ID := %sameServiceTwiceReady%);
      END_FBS
      SUBAPPS
        GetEndpointFromServiceRegistryEntry : GetEndpointFromServiceRegistryEntry;
        GetEndpointFromServiceRegistryEntry_1 : GetEndpointFromServiceRegistryEntry;
        RegisterService2 : RegisterServicePartialOpcUa(serviceURI := %serviceURI2%, version := %serviceVersion%, udp := false, metadata := %metadata%, SRendpoint := %serviceRegistryAddress%);
        RegisterService1 : RegisterServicePartialOpcUa(serviceURI := %serviceURI%, version := %serviceVersion%, udp := false, metadata := %metadata%, SRendpoint := %serviceRegistryAddress%);
        QueryServiceHTTPSub : QueryServiceOpcUaSub(version := %serviceVersion%, address := %serviceRegistryAddress%);
      END_SUBAPPS
      SUBAPPLICATION Sequencer
        EVENT_INPUT
          Next;
        END_EVENT
        EVENT_OUTPUT
          E0;
          E1;
          E2;
          E3;
          E4;
          E5;
          E6;
          E7;
          E8;
          E9;
          E10;
          E11;
        END_EVENT
      END_SUBAPPLICATION
      EVENT_CONNECTIONS
        Service1.CNF TO Sequencer.Next;
        FieldsToArrowheadSystem.CNF TO Service1.REQ;
        GET_AT_INDEX_1.CNF TO GetEndpointFromServiceRegistryEntry.REQ;
        GET_AT_INDEX.CNF TO GET_AT_INDEX_1.REQ;
        GetEndpointFromServiceRegistryEntry.CNF TO GetEndpointFromServiceRegistryEntry_1.REQ;
        GetEndpointFromServiceRegistryEntry_1.CNF TO Sequencer.Next;
        F_EQ_3.CNF TO F_EQ_2.REQ;
        F_EQ.CNF TO Service1RegisteredPos0.REQ;
        Sequencer.E3 TO F_EQ_3_1.REQ;
        F_EQ_3_1.CNF TO F_EQ_2_1.REQ;
        Sequencer.E6 TO F_EQ_1.REQ;
        F_EQ_1.CNF TO Service2RegisteredPos0.REQ;
        Sequencer.E9 TO F_EQ_1_1.REQ;
        F_EQ_1_1.CNF TO F_EQ_1_1_1.REQ;
        Service1RegisteredPos0.CNF TO F_EQ_4.REQ;
        F_EQ_4.CNF TO Service2NotRegisteredPos1.REQ;
        Service2RegisteredPos0.CNF TO F_EQ_4_1.REQ;
        F_EQ_4_1.CNF TO Service1NotRegisteredPos1.REQ;
        F_EQ_1_1_1.CNF TO F_AND.REQ;
        F_AND.CNF TO BothServicesNotRegistered.REQ;
        BothServicesRegistered.CNF TO E_MERGE.EI1;
        BothServicesNotRegistered.CNF TO E_MERGE.EI2;
        Service1NotRegisteredPos1.CNF TO E_MERGE.EI2;
        Service2NotRegisteredPos1.CNF TO E_MERGE.EI2;
        E_MERGE.EO TO Sequencer.Next;
        E_MERGE_1.EO TO Sequencer.Next;
        F_EQ_2_1.CNF TO F_AND_1.REQ;
        F_OR.CNF TO BothServicesRegistered.REQ;
        F_EQ_2.CNF TO F_AND_1_1.REQ;
        F_AND_1.CNF TO BOOL2BOOL.REQ;
        BOOL2BOOL.CNF TO F_EQ_3.REQ;
        F_AND_1_1.CNF TO BOOL2BOOL_1.REQ;
        BOOL2BOOL_1.CNF TO F_OR.REQ;
        SUBL_0.IND TO FieldsToArrowheadSystem_1.REQ;
        FieldsToArrowheadSystem_1.CNF TO FieldsToArrowheadSystem.REQ;
        START.COLD TO SUBL_0.INIT;
        START.WARM TO SUBL_0.INIT;
        Sequencer.E1 TO RegisterService2.register;
        Sequencer.E7 TO RegisterService2.unregister;
        RegisterService2.doneRegister TO E_MERGE_1.EI1;
        RegisterService2.doneUnregister TO E_MERGE_1.EI2;
        Sequencer.E0 TO RegisterService1.register;
        Sequencer.E4 TO RegisterService1.unregister;
        RegisterService1.doneRegister TO E_MERGE_1.EI1;
        RegisterService1.doneUnregister TO E_MERGE_1.EI2;
        Sequencer.E2 TO QueryServiceHTTPSub.REQ;
        Sequencer.E5 TO QueryServiceHTTPSub.REQ;
        Sequencer.E8 TO QueryServiceHTTPSub.REQ;
        QueryServiceHTTPSub.CNF TO GET_AT_INDEX.REQ;
        SUBL_0.INITO TO PUBL_0.INIT;
        Sequencer.E10 TO PUBL_0.REQ;
      END_CONNECTIONS
      DATA_CONNECTIONS
        GET_AT_INDEX.OUT TO GetEndpointFromServiceRegistryEntry.serviceRegistryEntry;
        GET_AT_INDEX_1.OUT TO GetEndpointFromServiceRegistryEntry_1.serviceRegistryEntry;
        GetEndpointFromServiceRegistryEntry_1.endpoint TO F_EQ_2.IN2;
        GetEndpointFromServiceRegistryEntry.endpoint TO F_EQ_3.IN2;
        GetEndpointFromServiceRegistryEntry.endpoint TO F_EQ.IN2;
        F_EQ.OUT TO Service1RegisteredPos0.check;
        GetEndpointFromServiceRegistryEntry_1.endpoint TO F_EQ_2_1.IN2;
        GetEndpointFromServiceRegistryEntry.endpoint TO F_EQ_3_1.IN2;
        GetEndpointFromServiceRegistryEntry.endpoint TO F_EQ_1.IN2;
        F_EQ_1.OUT TO Service2RegisteredPos0.check;
        GetEndpointFromServiceRegistryEntry.endpoint TO F_EQ_1_1.IN2;
        GetEndpointFromServiceRegistryEntry_1.endpoint TO F_EQ_1_1_1.IN2;
        GetEndpointFromServiceRegistryEntry_1.endpoint TO F_EQ_4.IN2;
        F_EQ_4.OUT TO Service2NotRegisteredPos1.check;
        GetEndpointFromServiceRegistryEntry_1.endpoint TO F_EQ_4_1.IN2;
        F_EQ_4_1.OUT TO Service1NotRegisteredPos1.check;
        F_EQ_1_1.OUT TO F_AND.IN1;
        F_EQ_1_1_1.OUT TO F_AND.IN2;
        F_AND.OUT TO BothServicesNotRegistered.check;
        F_EQ_3_1.OUT TO F_AND_1.IN1;
        F_EQ_2_1.OUT TO F_AND_1.IN2;
        F_OR.OUT TO BothServicesRegistered.check;
        F_EQ_3.OUT TO F_AND_1_1.IN1;
        F_EQ_2.OUT TO F_AND_1_1.IN2;
        F_AND_1.OUT TO BOOL2BOOL.IN;
        BOOL2BOOL.OUT TO F_OR.IN1;
        F_AND_1_1.OUT TO BOOL2BOOL_1.IN;
        BOOL2BOOL_1.OUT TO F_OR.IN2;
        Service1.arrowheadService TO RegisterService2.providedService;
        FieldsToArrowheadSystem_1.arrowheadSystem TO RegisterService2.provider;
        Service1.arrowheadService TO RegisterService1.providedService;
        FieldsToArrowheadSystem.arrowheadSystem TO RegisterService1.provider;
        Service1.arrowheadService TO QueryServiceHTTPSub.service;
        QueryServiceHTTPSub.serviceEntries TO GET_AT_INDEX.IN_ARRAY;
        QueryServiceHTTPSub.serviceEntries TO GET_AT_INDEX_1.IN_ARRAY;
      END_CONNECTIONS
    END_RESOURCE
    RESOURCE VersionInterfaceAndMetadata : EMB_RES
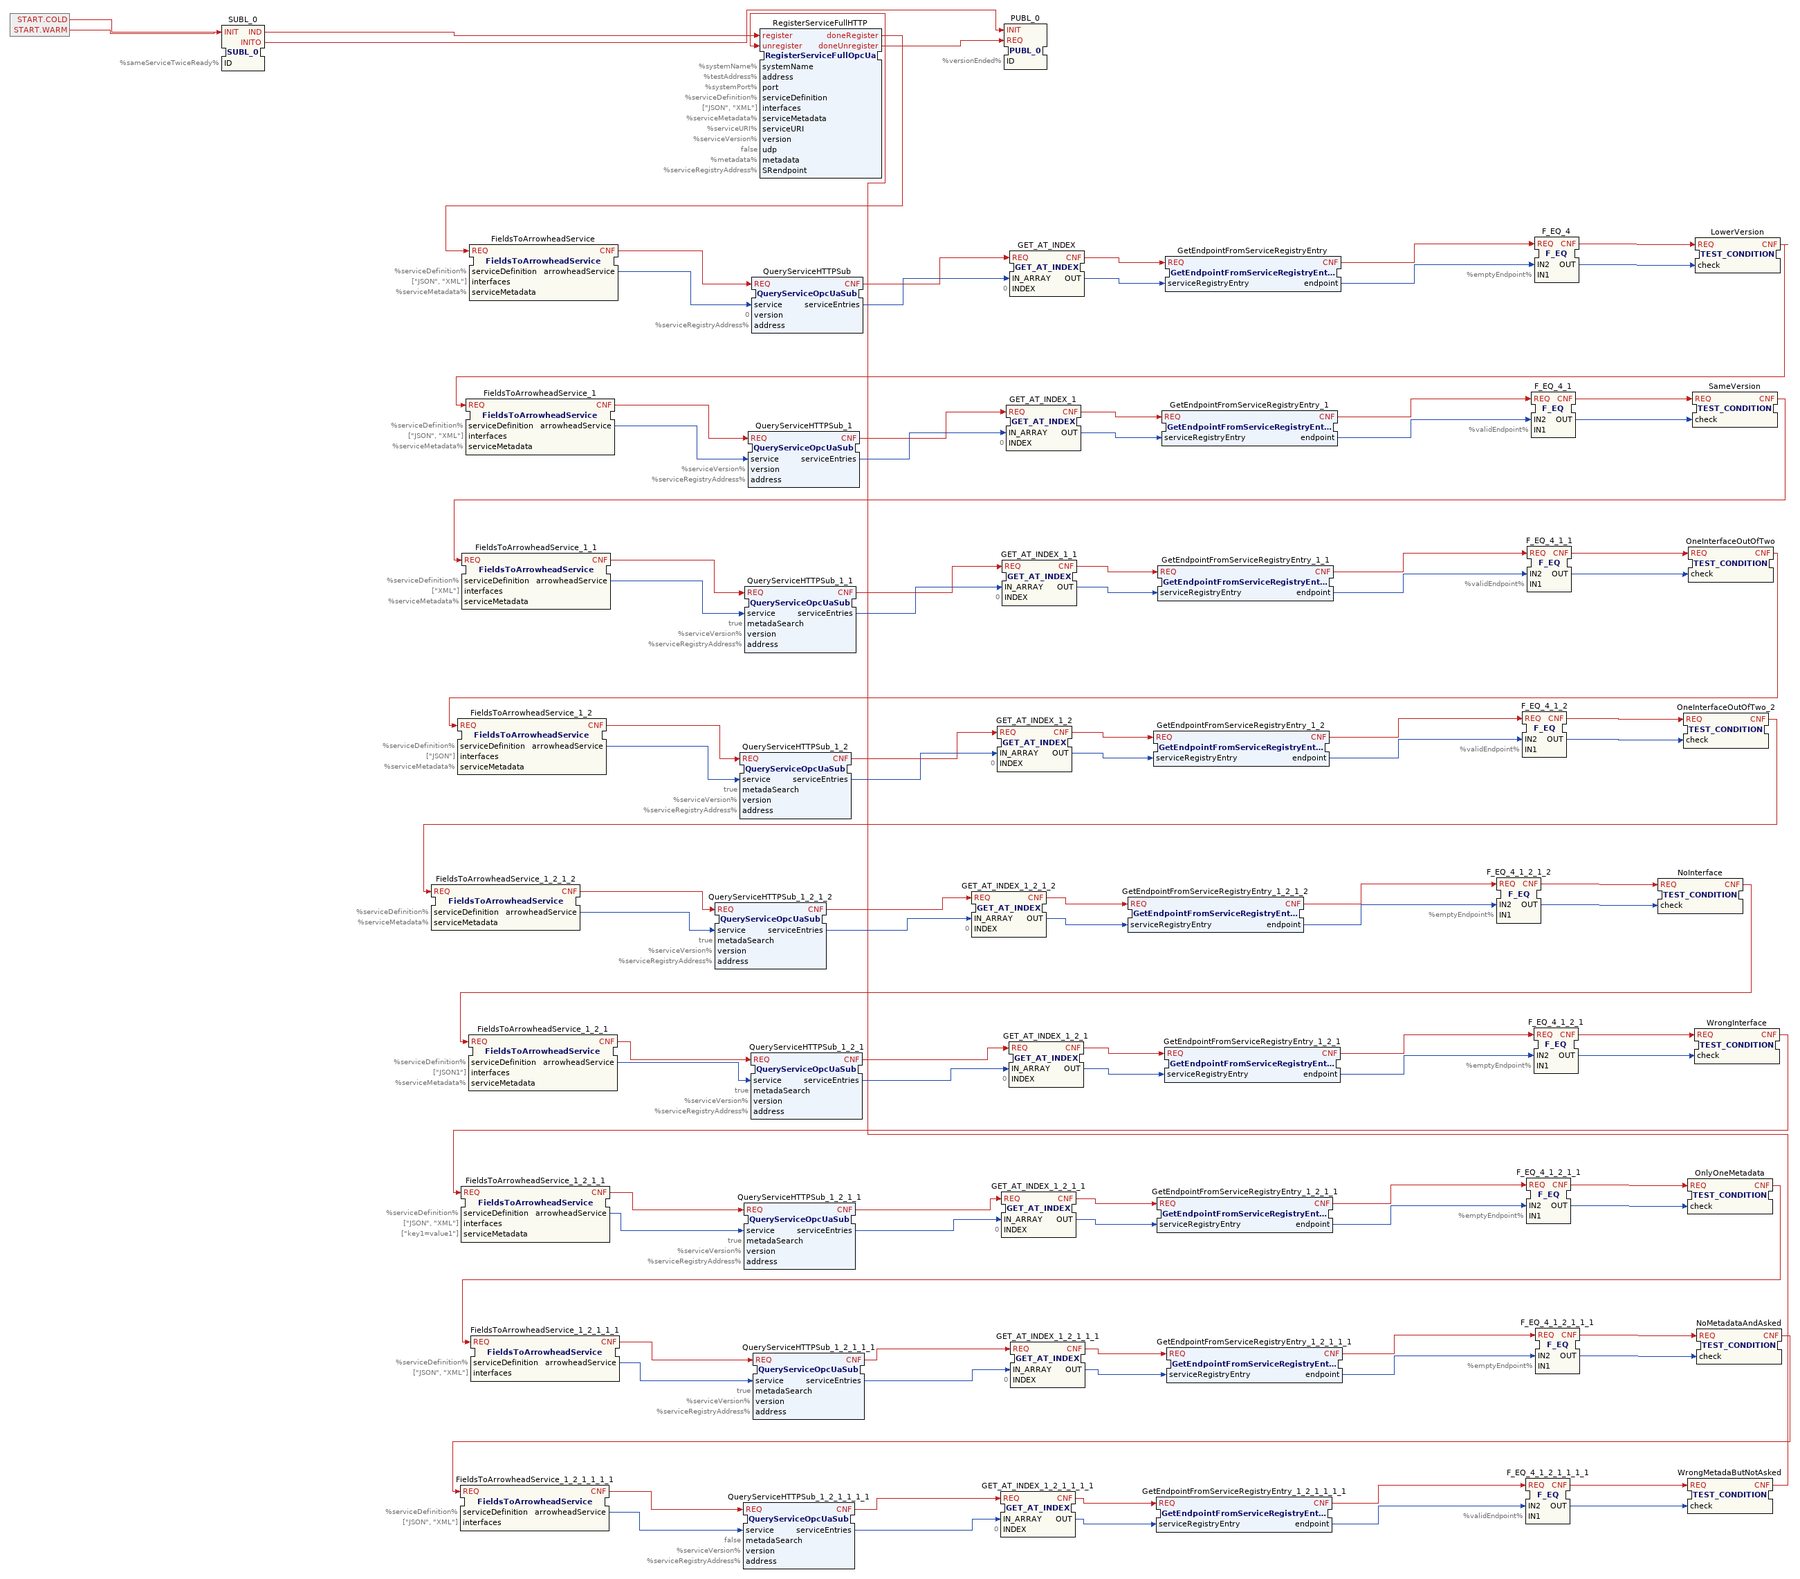
      FBS
        FieldsToArrowheadService : FieldsToArrowheadService(serviceDefinition := %serviceDefinition%, interfaces := ["JSON", "XML"], serviceMetadata := %serviceMetadata%);
        GET_AT_INDEX : GET_AT_INDEX(INDEX := 0);
        F_EQ_4 : F_EQ(IN1 := %emptyEndpoint%);
        LowerVersion : TEST_CONDITION;
        FieldsToArrowheadService_1 : FieldsToArrowheadService(serviceDefinition := %serviceDefinition%, interfaces := ["JSON", "XML"], serviceMetadata := %serviceMetadata%);
        SameVersion : TEST_CONDITION;
        GET_AT_INDEX_1 : GET_AT_INDEX(INDEX := 0);
        F_EQ_4_1 : F_EQ(IN1 := %validEndpoint%);
        OneInterfaceOutOfTwo : TEST_CONDITION;
        F_EQ_4_1_1 : F_EQ(IN1 := %validEndpoint%);
        FieldsToArrowheadService_1_1 : FieldsToArrowheadService(serviceDefinition := %serviceDefinition%, interfaces := ["XML"], serviceMetadata := %serviceMetadata%);
        GET_AT_INDEX_1_1 : GET_AT_INDEX(INDEX := 0);
        OneInterfaceOutOfTwo_2 : TEST_CONDITION;
        F_EQ_4_1_2 : F_EQ(IN1 := %validEndpoint%);
        FieldsToArrowheadService_1_2 : FieldsToArrowheadService(serviceDefinition := %serviceDefinition%, interfaces := ["JSON"], serviceMetadata := %serviceMetadata%);
        GET_AT_INDEX_1_2 : GET_AT_INDEX(INDEX := 0);
        WrongInterface : TEST_CONDITION;
        GET_AT_INDEX_1_2_1 : GET_AT_INDEX(INDEX := 0);
        FieldsToArrowheadService_1_2_1 : FieldsToArrowheadService(serviceDefinition := %serviceDefinition%, interfaces := ["JSON1"], serviceMetadata := %serviceMetadata%);
        F_EQ_4_1_2_1 : F_EQ(IN1 := %emptyEndpoint%);
        SUBL_0 : SUBL_0(ID := %sameServiceTwiceReady%);
        OnlyOneMetadata : TEST_CONDITION;
        F_EQ_4_1_2_1_1 : F_EQ(IN1 := %emptyEndpoint%);
        FieldsToArrowheadService_1_2_1_1 : FieldsToArrowheadService(serviceDefinition := %serviceDefinition%, interfaces := ["JSON", "XML"], serviceMetadata := ["key1=value1"]);
        GET_AT_INDEX_1_2_1_1 : GET_AT_INDEX(INDEX := 0);
        FieldsToArrowheadService_1_2_1_1_1 : FieldsToArrowheadService(serviceDefinition := %serviceDefinition%, interfaces := ["JSON", "XML"]);
        F_EQ_4_1_2_1_1_1 : F_EQ(IN1 := %emptyEndpoint%);
        GET_AT_INDEX_1_2_1_1_1 : GET_AT_INDEX(INDEX := 0);
        NoMetadataAndAsked : TEST_CONDITION;
        F_EQ_4_1_2_1_2 : F_EQ(IN1 := %emptyEndpoint%);
        GET_AT_INDEX_1_2_1_2 : GET_AT_INDEX(INDEX := 0);
        FieldsToArrowheadService_1_2_1_2 : FieldsToArrowheadService(serviceDefinition := %serviceDefinition%, serviceMetadata := %serviceMetadata%);
        NoInterface : TEST_CONDITION;
        GET_AT_INDEX_1_2_1_1_1_1 : GET_AT_INDEX(INDEX := 0);
        F_EQ_4_1_2_1_1_1_1 : F_EQ(IN1 := %validEndpoint%);
        WrongMetadaButNotAsked : TEST_CONDITION;
        FieldsToArrowheadService_1_2_1_1_1_1 : FieldsToArrowheadService(serviceDefinition := %serviceDefinition%, interfaces := ["JSON", "XML"]);
        PUBL_0 : PUBL_0(ID := %versionEnded%);
      END_FBS
      SUBAPPS
        GetEndpointFromServiceRegistryEntry : GetEndpointFromServiceRegistryEntry;
        GetEndpointFromServiceRegistryEntry_1 : GetEndpointFromServiceRegistryEntry;
        GetEndpointFromServiceRegistryEntry_1_1 : GetEndpointFromServiceRegistryEntry;
        GetEndpointFromServiceRegistryEntry_1_2 : GetEndpointFromServiceRegistryEntry;
        GetEndpointFromServiceRegistryEntry_1_2_1 : GetEndpointFromServiceRegistryEntry;
        GetEndpointFromServiceRegistryEntry_1_2_1_1 : GetEndpointFromServiceRegistryEntry;
        GetEndpointFromServiceRegistryEntry_1_2_1_1_1 : GetEndpointFromServiceRegistryEntry;
        GetEndpointFromServiceRegistryEntry_1_2_1_2 : GetEndpointFromServiceRegistryEntry;
        GetEndpointFromServiceRegistryEntry_1_2_1_1_1_1 : GetEndpointFromServiceRegistryEntry;
        RegisterServiceFullHTTP : RegisterServiceFullOpcUa(systemName := %systemName%, address := %testAddress%, port := %systemPort%, serviceDefinition := %serviceDefinition%, interfaces := ["JSON", "XML"], serviceMetadata := %serviceMetadata%, serviceURI := %serviceURI%, version := %serviceVersion%, udp := false, metadata := %metadata%, SRendpoint := %serviceRegistryAddress%);
        QueryServiceHTTPSub : QueryServiceOpcUaSub(version := 0, address := %serviceRegistryAddress%);
        QueryServiceHTTPSub_1 : QueryServiceOpcUaSub(version := %serviceVersion%, address := %serviceRegistryAddress%);
        QueryServiceHTTPSub_1_1 : QueryServiceOpcUaSub(metadaSearch := true, version := %serviceVersion%, address := %serviceRegistryAddress%);
        QueryServiceHTTPSub_1_2 : QueryServiceOpcUaSub(metadaSearch := true, version := %serviceVersion%, address := %serviceRegistryAddress%);
        QueryServiceHTTPSub_1_2_1_2 : QueryServiceOpcUaSub(metadaSearch := true, version := %serviceVersion%, address := %serviceRegistryAddress%);
        QueryServiceHTTPSub_1_2_1 : QueryServiceOpcUaSub(metadaSearch := true, version := %serviceVersion%, address := %serviceRegistryAddress%);
        QueryServiceHTTPSub_1_2_1_1 : QueryServiceOpcUaSub(metadaSearch := true, version := %serviceVersion%, address := %serviceRegistryAddress%);
        QueryServiceHTTPSub_1_2_1_1_1 : QueryServiceOpcUaSub(metadaSearch := true, version := %serviceVersion%, address := %serviceRegistryAddress%);
        QueryServiceHTTPSub_1_2_1_1_1_1 : QueryServiceOpcUaSub(metadaSearch := false, version := %serviceVersion%, address := %serviceRegistryAddress%);
      END_SUBAPPS
      EVENT_CONNECTIONS
        GET_AT_INDEX.CNF TO GetEndpointFromServiceRegistryEntry.REQ;
        GetEndpointFromServiceRegistryEntry.CNF TO F_EQ_4.REQ;
        F_EQ_4.CNF TO LowerVersion.REQ;
        LowerVersion.CNF TO FieldsToArrowheadService_1.REQ;
        GET_AT_INDEX_1.CNF TO GetEndpointFromServiceRegistryEntry_1.REQ;
        GetEndpointFromServiceRegistryEntry_1.CNF TO F_EQ_4_1.REQ;
        F_EQ_4_1.CNF TO SameVersion.REQ;
        GetEndpointFromServiceRegistryEntry_1_1.CNF TO F_EQ_4_1_1.REQ;
        F_EQ_4_1_1.CNF TO OneInterfaceOutOfTwo.REQ;
        SameVersion.CNF TO FieldsToArrowheadService_1_1.REQ;
        GET_AT_INDEX_1_1.CNF TO GetEndpointFromServiceRegistryEntry_1_1.REQ;
        GetEndpointFromServiceRegistryEntry_1_2.CNF TO F_EQ_4_1_2.REQ;
        F_EQ_4_1_2.CNF TO OneInterfaceOutOfTwo_2.REQ;
        OneInterfaceOutOfTwo.CNF TO FieldsToArrowheadService_1_2.REQ;
        GET_AT_INDEX_1_2.CNF TO GetEndpointFromServiceRegistryEntry_1_2.REQ;
        GET_AT_INDEX_1_2_1.CNF TO GetEndpointFromServiceRegistryEntry_1_2_1.REQ;
        GetEndpointFromServiceRegistryEntry_1_2_1.CNF TO F_EQ_4_1_2_1.REQ;
        F_EQ_4_1_2_1.CNF TO WrongInterface.REQ;
        GetEndpointFromServiceRegistryEntry_1_2_1_1.CNF TO F_EQ_4_1_2_1_1.REQ;
        F_EQ_4_1_2_1_1.CNF TO OnlyOneMetadata.REQ;
        WrongInterface.CNF TO FieldsToArrowheadService_1_2_1_1.REQ;
        GET_AT_INDEX_1_2_1_1.CNF TO GetEndpointFromServiceRegistryEntry_1_2_1_1.REQ;
        OnlyOneMetadata.CNF TO FieldsToArrowheadService_1_2_1_1_1.REQ;
        GetEndpointFromServiceRegistryEntry_1_2_1_1_1.CNF TO F_EQ_4_1_2_1_1_1.REQ;
        GET_AT_INDEX_1_2_1_1_1.CNF TO GetEndpointFromServiceRegistryEntry_1_2_1_1_1.REQ;
        F_EQ_4_1_2_1_1_1.CNF TO NoMetadataAndAsked.REQ;
        OneInterfaceOutOfTwo_2.CNF TO FieldsToArrowheadService_1_2_1_2.REQ;
        GET_AT_INDEX_1_2_1_2.CNF TO GetEndpointFromServiceRegistryEntry_1_2_1_2.REQ;
        GetEndpointFromServiceRegistryEntry_1_2_1_2.CNF TO F_EQ_4_1_2_1_2.REQ;
        F_EQ_4_1_2_1_2.CNF TO NoInterface.REQ;
        NoInterface.CNF TO FieldsToArrowheadService_1_2_1.REQ;
        GET_AT_INDEX_1_2_1_1_1_1.CNF TO GetEndpointFromServiceRegistryEntry_1_2_1_1_1_1.REQ;
        GetEndpointFromServiceRegistryEntry_1_2_1_1_1_1.CNF TO F_EQ_4_1_2_1_1_1_1.REQ;
        F_EQ_4_1_2_1_1_1_1.CNF TO WrongMetadaButNotAsked.REQ;
        NoMetadataAndAsked.CNF TO FieldsToArrowheadService_1_2_1_1_1_1.REQ;
        START.COLD TO SUBL_0.INIT;
        START.WARM TO SUBL_0.INIT;
        SUBL_0.IND TO RegisterServiceFullHTTP.register;
        WrongMetadaButNotAsked.CNF TO RegisterServiceFullHTTP.unregister;
        RegisterServiceFullHTTP.doneRegister TO FieldsToArrowheadService.REQ;
        FieldsToArrowheadService.CNF TO QueryServiceHTTPSub.REQ;
        QueryServiceHTTPSub.CNF TO GET_AT_INDEX.REQ;
        FieldsToArrowheadService_1.CNF TO QueryServiceHTTPSub_1.REQ;
        QueryServiceHTTPSub_1.CNF TO GET_AT_INDEX_1.REQ;
        FieldsToArrowheadService_1_1.CNF TO QueryServiceHTTPSub_1_1.REQ;
        QueryServiceHTTPSub_1_1.CNF TO GET_AT_INDEX_1_1.REQ;
        FieldsToArrowheadService_1_2.CNF TO QueryServiceHTTPSub_1_2.REQ;
        QueryServiceHTTPSub_1_2.CNF TO GET_AT_INDEX_1_2.REQ;
        FieldsToArrowheadService_1_2_1_2.CNF TO QueryServiceHTTPSub_1_2_1_2.REQ;
        QueryServiceHTTPSub_1_2_1_2.CNF TO GET_AT_INDEX_1_2_1_2.REQ;
        FieldsToArrowheadService_1_2_1.CNF TO QueryServiceHTTPSub_1_2_1.REQ;
        QueryServiceHTTPSub_1_2_1.CNF TO GET_AT_INDEX_1_2_1.REQ;
        FieldsToArrowheadService_1_2_1_1.CNF TO QueryServiceHTTPSub_1_2_1_1.REQ;
        QueryServiceHTTPSub_1_2_1_1.CNF TO GET_AT_INDEX_1_2_1_1.REQ;
        FieldsToArrowheadService_1_2_1_1_1.CNF TO QueryServiceHTTPSub_1_2_1_1_1.REQ;
        QueryServiceHTTPSub_1_2_1_1_1.CNF TO GET_AT_INDEX_1_2_1_1_1.REQ;
        FieldsToArrowheadService_1_2_1_1_1_1.CNF TO QueryServiceHTTPSub_1_2_1_1_1_1.REQ;
        QueryServiceHTTPSub_1_2_1_1_1_1.CNF TO GET_AT_INDEX_1_2_1_1_1_1.REQ;
        SUBL_0.INITO TO PUBL_0.INIT;
        RegisterServiceFullHTTP.doneUnregister TO PUBL_0.REQ;
      END_CONNECTIONS
      DATA_CONNECTIONS
        GET_AT_INDEX.OUT TO GetEndpointFromServiceRegistryEntry.serviceRegistryEntry;
        GetEndpointFromServiceRegistryEntry.endpoint TO F_EQ_4.IN2;
        F_EQ_4.OUT TO LowerVersion.check;
        GET_AT_INDEX_1.OUT TO GetEndpointFromServiceRegistryEntry_1.serviceRegistryEntry;
        GetEndpointFromServiceRegistryEntry_1.endpoint TO F_EQ_4_1.IN2;
        F_EQ_4_1.OUT TO SameVersion.check;
        GetEndpointFromServiceRegistryEntry_1_1.endpoint TO F_EQ_4_1_1.IN2;
        F_EQ_4_1_1.OUT TO OneInterfaceOutOfTwo.check;
        GET_AT_INDEX_1_1.OUT TO GetEndpointFromServiceRegistryEntry_1_1.serviceRegistryEntry;
        GetEndpointFromServiceRegistryEntry_1_2.endpoint TO F_EQ_4_1_2.IN2;
        F_EQ_4_1_2.OUT TO OneInterfaceOutOfTwo_2.check;
        GET_AT_INDEX_1_2.OUT TO GetEndpointFromServiceRegistryEntry_1_2.serviceRegistryEntry;
        GET_AT_INDEX_1_2_1.OUT TO GetEndpointFromServiceRegistryEntry_1_2_1.serviceRegistryEntry;
        GetEndpointFromServiceRegistryEntry_1_2_1.endpoint TO F_EQ_4_1_2_1.IN2;
        F_EQ_4_1_2_1.OUT TO WrongInterface.check;
        GetEndpointFromServiceRegistryEntry_1_2_1_1.endpoint TO F_EQ_4_1_2_1_1.IN2;
        F_EQ_4_1_2_1_1.OUT TO OnlyOneMetadata.check;
        GET_AT_INDEX_1_2_1_1.OUT TO GetEndpointFromServiceRegistryEntry_1_2_1_1.serviceRegistryEntry;
        GetEndpointFromServiceRegistryEntry_1_2_1_1_1.endpoint TO F_EQ_4_1_2_1_1_1.IN2;
        GET_AT_INDEX_1_2_1_1_1.OUT TO GetEndpointFromServiceRegistryEntry_1_2_1_1_1.serviceRegistryEntry;
        F_EQ_4_1_2_1_1_1.OUT TO NoMetadataAndAsked.check;
        GET_AT_INDEX_1_2_1_2.OUT TO GetEndpointFromServiceRegistryEntry_1_2_1_2.serviceRegistryEntry;
        GetEndpointFromServiceRegistryEntry_1_2_1_2.endpoint TO F_EQ_4_1_2_1_2.IN2;
        F_EQ_4_1_2_1_2.OUT TO NoInterface.check;
        GET_AT_INDEX_1_2_1_1_1_1.OUT TO GetEndpointFromServiceRegistryEntry_1_2_1_1_1_1.serviceRegistryEntry;
        GetEndpointFromServiceRegistryEntry_1_2_1_1_1_1.endpoint TO F_EQ_4_1_2_1_1_1_1.IN2;
        F_EQ_4_1_2_1_1_1_1.OUT TO WrongMetadaButNotAsked.check;
        FieldsToArrowheadService.arrowheadService TO QueryServiceHTTPSub.service;
        QueryServiceHTTPSub.serviceEntries TO GET_AT_INDEX.IN_ARRAY;
        FieldsToArrowheadService_1.arrowheadService TO QueryServiceHTTPSub_1.service;
        QueryServiceHTTPSub_1.serviceEntries TO GET_AT_INDEX_1.IN_ARRAY;
        FieldsToArrowheadService_1_1.arrowheadService TO QueryServiceHTTPSub_1_1.service;
        QueryServiceHTTPSub_1_1.serviceEntries TO GET_AT_INDEX_1_1.IN_ARRAY;
        FieldsToArrowheadService_1_2.arrowheadService TO QueryServiceHTTPSub_1_2.service;
        QueryServiceHTTPSub_1_2.serviceEntries TO GET_AT_INDEX_1_2.IN_ARRAY;
        FieldsToArrowheadService_1_2_1_2.arrowheadService TO QueryServiceHTTPSub_1_2_1_2.service;
        QueryServiceHTTPSub_1_2_1_2.serviceEntries TO GET_AT_INDEX_1_2_1_2.IN_ARRAY;
        FieldsToArrowheadService_1_2_1.arrowheadService TO QueryServiceHTTPSub_1_2_1.service;
        QueryServiceHTTPSub_1_2_1.serviceEntries TO GET_AT_INDEX_1_2_1.IN_ARRAY;
        FieldsToArrowheadService_1_2_1_1.arrowheadService TO QueryServiceHTTPSub_1_2_1_1.service;
        QueryServiceHTTPSub_1_2_1_1.serviceEntries TO GET_AT_INDEX_1_2_1_1.IN_ARRAY;
        FieldsToArrowheadService_1_2_1_1_1.arrowheadService TO QueryServiceHTTPSub_1_2_1_1_1.service;
        QueryServiceHTTPSub_1_2_1_1_1.serviceEntries TO GET_AT_INDEX_1_2_1_1_1.IN_ARRAY;
        FieldsToArrowheadService_1_2_1_1_1_1.arrowheadService TO QueryServiceHTTPSub_1_2_1_1_1_1.service;
        QueryServiceHTTPSub_1_2_1_1_1_1.serviceEntries TO GET_AT_INDEX_1_2_1_1_1_1.IN_ARRAY;
      END_CONNECTIONS
    END_RESOURCE
    RESOURCE RegisterMoreServicesSubApp : EMB_RES
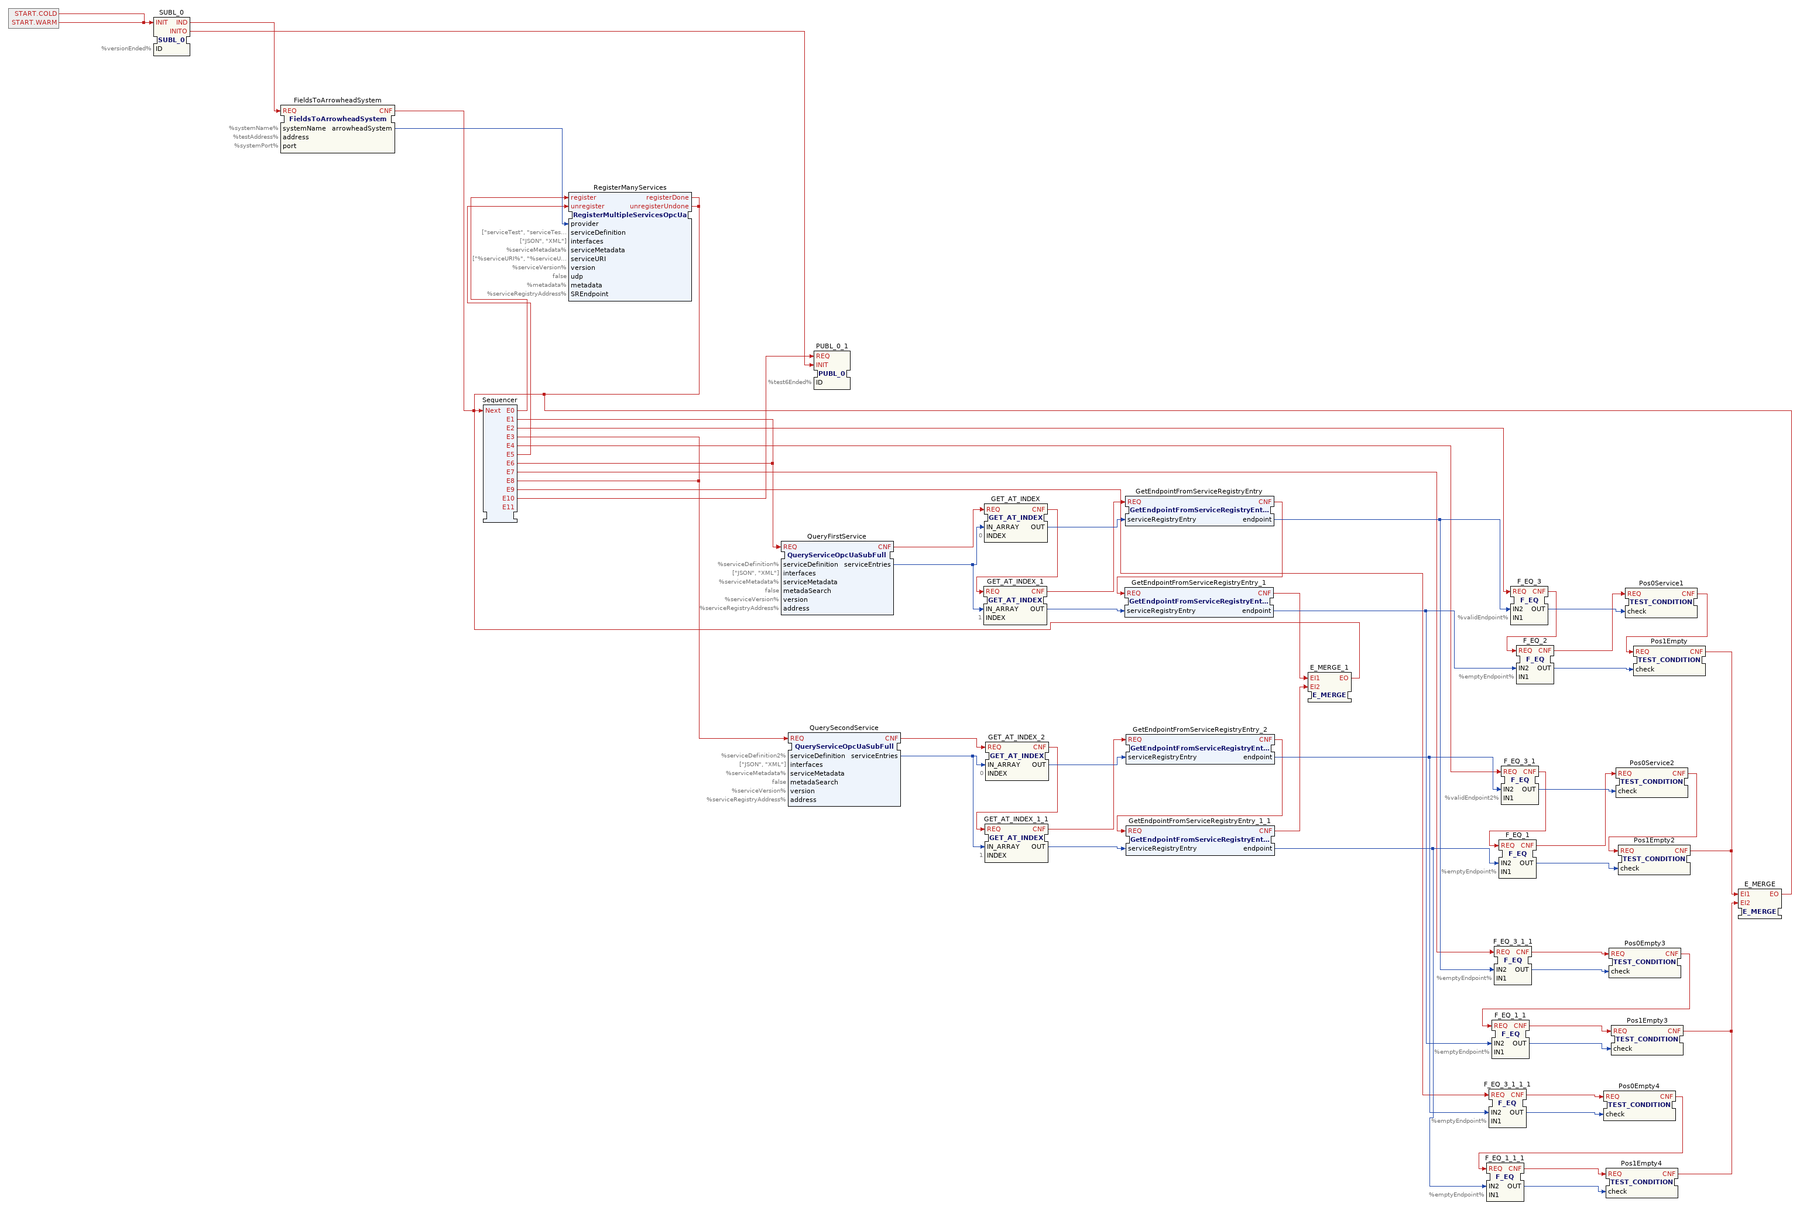
      FBS
        SUBL_0 : SUBL_0(ID := %versionEnded%);
        GET_AT_INDEX_1 : GET_AT_INDEX(INDEX := 1);
        FieldsToArrowheadSystem : FieldsToArrowheadSystem(systemName := %systemName%, address := %testAddress%, port := %systemPort%);
        F_EQ_2 : F_EQ(IN1 := %emptyEndpoint%);
        GET_AT_INDEX : GET_AT_INDEX(INDEX := 0);
        Pos1Empty2 : TEST_CONDITION;
        F_EQ_1 : F_EQ(IN1 := %emptyEndpoint%);
        Pos1Empty : TEST_CONDITION;
        GET_AT_INDEX_1_1 : GET_AT_INDEX(INDEX := 1);
        GET_AT_INDEX_2 : GET_AT_INDEX(INDEX := 0);
        Pos0Service1 : TEST_CONDITION;
        F_EQ_3 : F_EQ(IN1 := %validEndpoint%);
        F_EQ_3_1 : F_EQ(IN1 := %validEndpoint2%);
        Pos0Service2 : TEST_CONDITION;
        PUBL_0_1 : PUBL_0(ID := %test6Ended%);
        F_EQ_1_1 : F_EQ(IN1 := %emptyEndpoint%);
        F_EQ_3_1_1 : F_EQ(IN1 := %emptyEndpoint%);
        Pos1Empty3 : TEST_CONDITION;
        Pos0Empty3 : TEST_CONDITION;
        F_EQ_1_1_1 : F_EQ(IN1 := %emptyEndpoint%);
        Pos0Empty4 : TEST_CONDITION;
        Pos1Empty4 : TEST_CONDITION;
        F_EQ_3_1_1_1 : F_EQ(IN1 := %emptyEndpoint%);
        E_MERGE : E_MERGE;
        E_MERGE_1 : E_MERGE;
      END_FBS
      SUBAPPS
        GetEndpointFromServiceRegistryEntry_1 : GetEndpointFromServiceRegistryEntry;
        GetEndpointFromServiceRegistryEntry : GetEndpointFromServiceRegistryEntry;
        GetEndpointFromServiceRegistryEntry_1_1 : GetEndpointFromServiceRegistryEntry;
        GetEndpointFromServiceRegistryEntry_2 : GetEndpointFromServiceRegistryEntry;
        RegisterManyServices : RegisterMultipleServicesOpcUa(serviceDefinition := ["serviceTest", "serviceTest2"], interfaces := ["JSON", "XML"], serviceMetadata := %serviceMetadata%, serviceURI := ["%serviceURI%", "%serviceURI2%"], version := %serviceVersion%, udp := false, metadata := %metadata%, SREndpoint := %serviceRegistryAddress%);
        QueryFirstService : QueryServiceOpcUaSubFull(serviceDefinition := %serviceDefinition%, interfaces := ["JSON", "XML"], serviceMetadata := %serviceMetadata%, metadaSearch := false, version := %serviceVersion%, address := %serviceRegistryAddress%);
        QuerySecondService : QueryServiceOpcUaSubFull(serviceDefinition := %serviceDefinition2%, interfaces := ["JSON", "XML"], serviceMetadata := %serviceMetadata%, metadaSearch := false, version := %serviceVersion%, address := %serviceRegistryAddress%);
      END_SUBAPPS
      SUBAPPLICATION Sequencer
        EVENT_INPUT
          Next;
        END_EVENT
        EVENT_OUTPUT
          E0;
          E1;
          E2;
          E3;
          E4;
          E5;
          E6;
          E7;
          E8;
          E9;
          E10;
          E11;
        END_EVENT
      END_SUBAPPLICATION
      EVENT_CONNECTIONS
        GET_AT_INDEX_1.CNF TO GetEndpointFromServiceRegistryEntry.REQ;
        GetEndpointFromServiceRegistryEntry.CNF TO GetEndpointFromServiceRegistryEntry_1.REQ;
        SUBL_0.IND TO FieldsToArrowheadSystem.REQ;
        GET_AT_INDEX.CNF TO GET_AT_INDEX_1.REQ;
        FieldsToArrowheadSystem.CNF TO Sequencer.Next;
        GET_AT_INDEX_1_1.CNF TO GetEndpointFromServiceRegistryEntry_2.REQ;
        GetEndpointFromServiceRegistryEntry_2.CNF TO GetEndpointFromServiceRegistryEntry_1_1.REQ;
        GET_AT_INDEX_2.CNF TO GET_AT_INDEX_1_1.REQ;
        F_EQ_2.CNF TO Pos0Service1.REQ;
        Pos0Service1.CNF TO Pos1Empty.REQ;
        Sequencer.E2 TO F_EQ_3.REQ;
        F_EQ_3.CNF TO F_EQ_2.REQ;
        Sequencer.E4 TO F_EQ_3_1.REQ;
        F_EQ_3_1.CNF TO F_EQ_1.REQ;
        F_EQ_1.CNF TO Pos0Service2.REQ;
        Pos0Service2.CNF TO Pos1Empty2.REQ;
        Sequencer.E7 TO F_EQ_3_1_1.REQ;
        F_EQ_1_1.CNF TO Pos1Empty3.REQ;
        F_EQ_3_1_1.CNF TO Pos0Empty3.REQ;
        Pos0Empty3.CNF TO F_EQ_1_1.REQ;
        Pos0Empty4.CNF TO F_EQ_1_1_1.REQ;
        F_EQ_1_1_1.CNF TO Pos1Empty4.REQ;
        Sequencer.E9 TO F_EQ_3_1_1_1.REQ;
        F_EQ_3_1_1_1.CNF TO Pos0Empty4.REQ;
        Pos1Empty.CNF TO E_MERGE.EI1;
        Pos1Empty2.CNF TO E_MERGE.EI1;
        Pos1Empty3.CNF TO E_MERGE.EI2;
        Pos1Empty4.CNF TO E_MERGE.EI2;
        E_MERGE.EO TO Sequencer.Next;
        GetEndpointFromServiceRegistryEntry_1.CNF TO E_MERGE_1.EI1;
        GetEndpointFromServiceRegistryEntry_1_1.CNF TO E_MERGE_1.EI2;
        E_MERGE_1.EO TO Sequencer.Next;
        START.COLD TO SUBL_0.INIT;
        START.WARM TO SUBL_0.INIT;
        Sequencer.E0 TO RegisterManyServices.register;
        Sequencer.E5 TO RegisterManyServices.unregister;
        RegisterManyServices.registerDone TO Sequencer.Next;
        RegisterManyServices.unregisterUndone TO Sequencer.Next;
        Sequencer.E1 TO QueryFirstService.REQ;
        Sequencer.E6 TO QueryFirstService.REQ;
        QueryFirstService.CNF TO GET_AT_INDEX.REQ;
        Sequencer.E3 TO QuerySecondService.REQ;
        Sequencer.E8 TO QuerySecondService.REQ;
        QuerySecondService.CNF TO GET_AT_INDEX_2.REQ;
        Sequencer.E10 TO PUBL_0_1.REQ;
        SUBL_0.INITO TO PUBL_0_1.INIT;
      END_CONNECTIONS
      DATA_CONNECTIONS
        GET_AT_INDEX_1.OUT TO GetEndpointFromServiceRegistryEntry_1.serviceRegistryEntry;
        GetEndpointFromServiceRegistryEntry_1.endpoint TO F_EQ_2.IN2;
        GET_AT_INDEX.OUT TO GetEndpointFromServiceRegistryEntry.serviceRegistryEntry;
        F_EQ_1.OUT TO Pos1Empty2.check;
        F_EQ_2.OUT TO Pos1Empty.check;
        GET_AT_INDEX_1_1.OUT TO GetEndpointFromServiceRegistryEntry_1_1.serviceRegistryEntry;
        GetEndpointFromServiceRegistryEntry_1_1.endpoint TO F_EQ_1.IN2;
        GET_AT_INDEX_2.OUT TO GetEndpointFromServiceRegistryEntry_2.serviceRegistryEntry;
        GetEndpointFromServiceRegistryEntry.endpoint TO F_EQ_3.IN2;
        F_EQ_3.OUT TO Pos0Service1.check;
        GetEndpointFromServiceRegistryEntry_2.endpoint TO F_EQ_3_1.IN2;
        F_EQ_3_1.OUT TO Pos0Service2.check;
        GetEndpointFromServiceRegistryEntry_1.endpoint TO F_EQ_1_1.IN2;
        GetEndpointFromServiceRegistryEntry.endpoint TO F_EQ_3_1_1.IN2;
        F_EQ_1_1.OUT TO Pos1Empty3.check;
        F_EQ_3_1_1.OUT TO Pos0Empty3.check;
        GetEndpointFromServiceRegistryEntry_1_1.endpoint TO F_EQ_1_1_1.IN2;
        F_EQ_1_1_1.OUT TO Pos1Empty4.check;
        GetEndpointFromServiceRegistryEntry_2.endpoint TO F_EQ_3_1_1_1.IN2;
        F_EQ_3_1_1_1.OUT TO Pos0Empty4.check;
        FieldsToArrowheadSystem.arrowheadSystem TO RegisterManyServices.provider;
        QueryFirstService.serviceEntries TO GET_AT_INDEX_1.IN_ARRAY;
        QueryFirstService.serviceEntries TO GET_AT_INDEX.IN_ARRAY;
        QuerySecondService.serviceEntries TO GET_AT_INDEX_1_1.IN_ARRAY;
        QuerySecondService.serviceEntries TO GET_AT_INDEX_2.IN_ARRAY;
      END_CONNECTIONS
    END_RESOURCE
    RESOURCE OrchestratorNoRule : EMB_RES
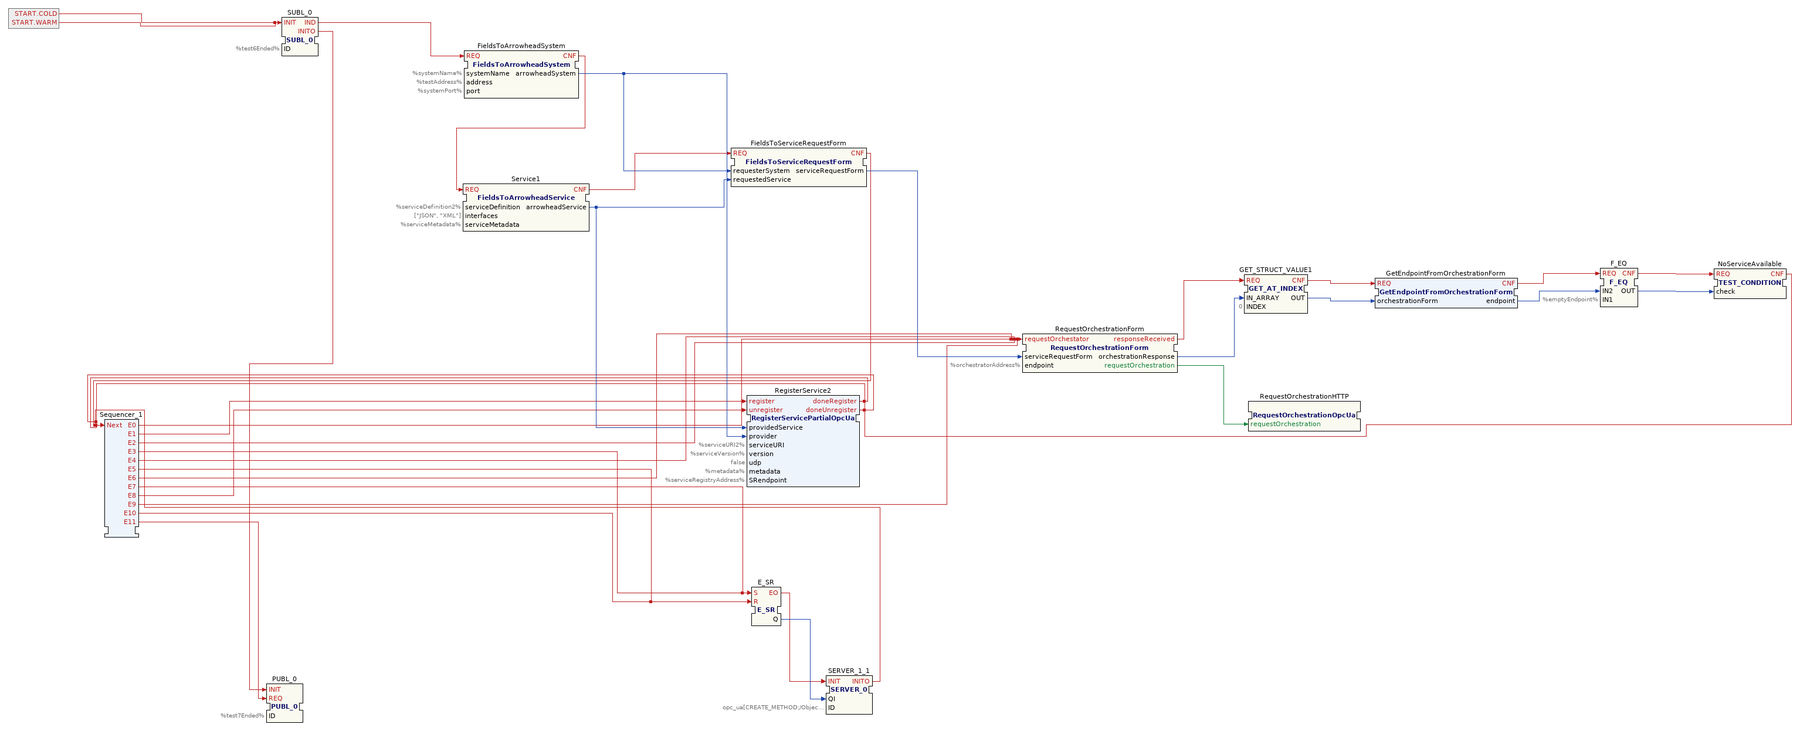
      FBS
        FieldsToServiceRequestForm : FieldsToServiceRequestForm;
        FieldsToArrowheadSystem : FieldsToArrowheadSystem(systemName := %systemName%, address := %testAddress%, port := %systemPort%);
        Service1 : FieldsToArrowheadService(serviceDefinition := %serviceDefinition2%, interfaces := ["JSON", "XML"], serviceMetadata := %serviceMetadata%);
        F_EQ : F_EQ(IN1 := %emptyEndpoint%);
        NoServiceAvailable : TEST_CONDITION;
        E_SR : E_SR;
        SUBL_0 : SUBL_0(ID := %test6Ended%);
        PUBL_0 : PUBL_0(ID := %test7Ended%);
        GET_STRUCT_VALUE1 : GET_AT_INDEX(INDEX := 0);
        RequestOrchestrationForm : RequestOrchestrationForm(endpoint := %orchestratorAddress%);
        RequestOrchestrationHTTP : RequestOrchestrationOpcUa;
        SERVER_1_1 : SERVER_0(ID := opc_ua[CREATE_METHOD;/Objects/serviceTest/start2]);
      END_FBS
      SUBAPPS
        GetEndpointFromOrchestrationForm : GetEndpointFromOrchestrationForm;
        RegisterService2 : RegisterServicePartialOpcUa(serviceURI := %serviceURI2%, version := %serviceVersion%, udp := false, metadata := %metadata%, SRendpoint := %serviceRegistryAddress%);
      END_SUBAPPS
      SUBAPPLICATION Sequencer_1
        EVENT_INPUT
          Next;
        END_EVENT
        EVENT_OUTPUT
          E0;
          E1;
          E2;
          E3;
          E4;
          E5;
          E6;
          E7;
          E8;
          E9;
          E10;
          E11;
        END_EVENT
      END_SUBAPPLICATION
      EVENT_CONNECTIONS
        FieldsToArrowheadSystem.CNF TO Service1.REQ;
        Service1.CNF TO FieldsToServiceRequestForm.REQ;
        GetEndpointFromOrchestrationForm.CNF TO F_EQ.REQ;
        F_EQ.CNF TO NoServiceAvailable.REQ;
        SUBL_0.IND TO FieldsToArrowheadSystem.REQ;
        GET_STRUCT_VALUE1.CNF TO GetEndpointFromOrchestrationForm.REQ;
        NoServiceAvailable.CNF TO Sequencer_1.Next;
        FieldsToServiceRequestForm.CNF TO Sequencer_1.Next;
        Sequencer_1.E3 TO E_SR.S;
        Sequencer_1.E5 TO E_SR.R;
        Sequencer_1.E7 TO E_SR.S;
        Sequencer_1.E10 TO E_SR.R;
        Sequencer_1.E0 TO RequestOrchestrationForm.requestOrchestator;
        Sequencer_1.E2 TO RequestOrchestrationForm.requestOrchestator;
        Sequencer_1.E4 TO RequestOrchestrationForm.requestOrchestator;
        Sequencer_1.E6 TO RequestOrchestrationForm.requestOrchestator;
        Sequencer_1.E9 TO RequestOrchestrationForm.requestOrchestator;
        RequestOrchestrationForm.responseReceived TO GET_STRUCT_VALUE1.REQ;
        START.COLD TO SUBL_0.INIT;
        START.WARM TO SUBL_0.INIT;
        Sequencer_1.E1 TO RegisterService2.register;
        Sequencer_1.E8 TO RegisterService2.unregister;
        RegisterService2.doneRegister TO Sequencer_1.Next;
        RegisterService2.doneUnregister TO Sequencer_1.Next;
        E_SR.EO TO SERVER_1_1.INIT;
        SERVER_1_1.INITO TO Sequencer_1.Next;
        SUBL_0.INITO TO PUBL_0.INIT;
        Sequencer_1.E11 TO PUBL_0.REQ;
      END_CONNECTIONS
      DATA_CONNECTIONS
        FieldsToArrowheadSystem.arrowheadSystem TO FieldsToServiceRequestForm.requesterSystem;
        Service1.arrowheadService TO FieldsToServiceRequestForm.requestedService;
        GetEndpointFromOrchestrationForm.endpoint TO F_EQ.IN2;
        F_EQ.OUT TO NoServiceAvailable.check;
        GET_STRUCT_VALUE1.OUT TO GetEndpointFromOrchestrationForm.orchestrationForm;
        FieldsToServiceRequestForm.serviceRequestForm TO RequestOrchestrationForm.serviceRequestForm;
        RequestOrchestrationForm.orchestrationResponse TO GET_STRUCT_VALUE1.IN_ARRAY;
        Service1.arrowheadService TO RegisterService2.providedService;
        FieldsToArrowheadSystem.arrowheadSystem TO RegisterService2.provider;
        E_SR.Q TO SERVER_1_1.QI;
      END_CONNECTIONS
      ADAPTER_CONNECTIONS
        RequestOrchestrationForm.requestOrchestration TO RequestOrchestrationHTTP.requestOrchestration;
      END_CONNECTIONS
    END_RESOURCE
    RESOURCE OrchestrationWithRules : EMB_RES
      FBS
        FieldsToArrowheadSystem : FieldsToArrowheadSystem(systemName := %systemName%, address := %testAddress%, port := %systemPort%);
        Service1 : FieldsToArrowheadService(serviceDefinition := %serviceDefinition%, interfaces := ["JSON", "XML"], serviceMetadata := %serviceMetadata%);
        F_EQ : F_EQ(IN1 := %emptyEndpoint%);
        NoServiceAvailable : TEST_CONDITION;
        E_SR : E_SR;
        SUBL_0 : SUBL_0(ID := %test7Ended%);
        PUBL_0 : PUBL_0(ID := %test8Ended%);
        F_EQ_1 : F_EQ(IN1 := %validEndpoint%);
        ServiceAvailable : TEST_CONDITION;
        E_SR_1 : E_SR;
        E_SWITCH : E_SWITCH;
        SERVER_1_1 : SERVER_0(ID := opc_ua[CREATE_METHOD;/Objects/serviceTest/start2]);
        E_DELAY : E_DELAY(DT := T#1s);
        E_DELAY_1 : E_DELAY(DT := T#1s);
        STRING2STRING_3_1 : STRING2STRING(IN := STRING#%orchRuleData%);
        STRING2STRING_3 : STRING2STRING(IN := STRING#%authRuleData%);
        CLIENT_1_2 : CLIENT_1_0(QI := 1, ID := opc_ua[CALL_METHOD; %authRuleEndpoint%#; /Objects/2:Authorization/2:addSystemToAuthorized]);
        CLIENT_1_2_1 : CLIENT_1_0(QI := 1, ID := opc_ua[CALL_METHOD; %orchestratorEndpoint%#; /Objects/2:Orchestrator/2:store]);
      END_FBS
      SUBAPPS
        RegisterService2 : RegisterServicePartialOpcUa(serviceURI := %serviceURI%, version := %serviceVersion%, udp := false, metadata := %metadata%, SRendpoint := %serviceRegistryAddress%);
        GetEndpointFromOrchestrationHTTPPFull : GetEndpointFromOrchestrationOpcUaFull(systemName := %systemName%, address := %testAddress%, port := %systemPort%, serviceDefinition := %serviceDefinition%, interfaces := ["JSON", "XML"], serviceMetadata := %serviceMetadata%, orchestratorEndpoint := %orchestratorAddress%, INDEX := 0);
      END_SUBAPPS
      SUBAPPLICATION Sequencer_1
        EVENT_INPUT
          Next;
        END_EVENT
        EVENT_OUTPUT
          E0;
          E1;
          E2;
          E3;
          E4;
          E5;
          E6;
          E7;
          E8;
          E9;
          E10;
          E11;
          E12;
          E13;
          E14;
          E15;
        END_EVENT
      END_SUBAPPLICATION
      EVENT_CONNECTIONS
        FieldsToArrowheadSystem.CNF TO Service1.REQ;
        F_EQ.CNF TO NoServiceAvailable.REQ;
        SUBL_0.IND TO FieldsToArrowheadSystem.REQ;
        NoServiceAvailable.CNF TO Sequencer_1.Next;
        Service1.CNF TO Sequencer_1.Next;
        Sequencer_1.E5 TO E_SR.S;
        Sequencer_1.E10 TO E_SR.R;
        F_EQ_1.CNF TO ServiceAvailable.REQ;
        ServiceAvailable.CNF TO Sequencer_1.Next;
        Sequencer_1.E3 TO E_SR_1.S;
        Sequencer_1.E8 TO E_SR_1.R;
        E_SR_1.EO TO Sequencer_1.Next;
        E_SWITCH.EO0 TO F_EQ.REQ;
        E_SWITCH.EO1 TO F_EQ_1.REQ;
        START.WARM TO SUBL_0.INIT;
        START.COLD TO SUBL_0.INIT;
        Sequencer_1.E2 TO RegisterService2.register;
        Sequencer_1.E7 TO RegisterService2.unregister;
        RegisterService2.doneRegister TO Sequencer_1.Next;
        RegisterService2.doneUnregister TO Sequencer_1.Next;
        Sequencer_1.E11 TO GetEndpointFromOrchestrationHTTPPFull.REQ;
        Sequencer_1.E9 TO GetEndpointFromOrchestrationHTTPPFull.REQ;
        Sequencer_1.E6 TO GetEndpointFromOrchestrationHTTPPFull.REQ;
        Sequencer_1.E4 TO GetEndpointFromOrchestrationHTTPPFull.REQ;
        Sequencer_1.E1 TO GetEndpointFromOrchestrationHTTPPFull.REQ;
        GetEndpointFromOrchestrationHTTPPFull.CNF TO E_SWITCH.EI;
        SUBL_0.INITO TO PUBL_0.INIT;
        Sequencer_1.E12 TO PUBL_0.REQ;
        Sequencer_1.E0 TO STRING2STRING_3.REQ;
        E_SR.EO TO Sequencer_1.Next;
        STRING2STRING_3.CNF TO CLIENT_1_2.INIT;
        E_DELAY.EO TO CLIENT_1_2.REQ;
        CLIENT_1_2.INITO TO E_DELAY.START;
        CLIENT_1_2.CNF TO STRING2STRING_3_1.REQ;
        STRING2STRING_3_1.CNF TO CLIENT_1_2_1.INIT;
        E_DELAY_1.EO TO CLIENT_1_2_1.REQ;
        CLIENT_1_2_1.INITO TO E_DELAY_1.START;
        CLIENT_1_2_1.CNF TO Sequencer_1.Next;
      END_CONNECTIONS
      DATA_CONNECTIONS
        F_EQ.OUT TO NoServiceAvailable.check;
        F_EQ_1.OUT TO ServiceAvailable.check;
        E_SR_1.Q TO E_SWITCH.G;
        E_SR.Q TO SERVER_1_1.QI;
        Service1.arrowheadService TO RegisterService2.providedService;
        FieldsToArrowheadSystem.arrowheadSystem TO RegisterService2.provider;
        GetEndpointFromOrchestrationHTTPPFull.endpoint TO F_EQ_1.IN2;
        GetEndpointFromOrchestrationHTTPPFull.endpoint TO F_EQ.IN2;
        STRING2STRING_3.OUT TO CLIENT_1_2.SD_1;
        STRING2STRING_3_1.OUT TO CLIENT_1_2_1.SD_1;
      END_CONNECTIONS
    END_RESOURCE
    RESOURCE PublishSubscribe : EMB_RES
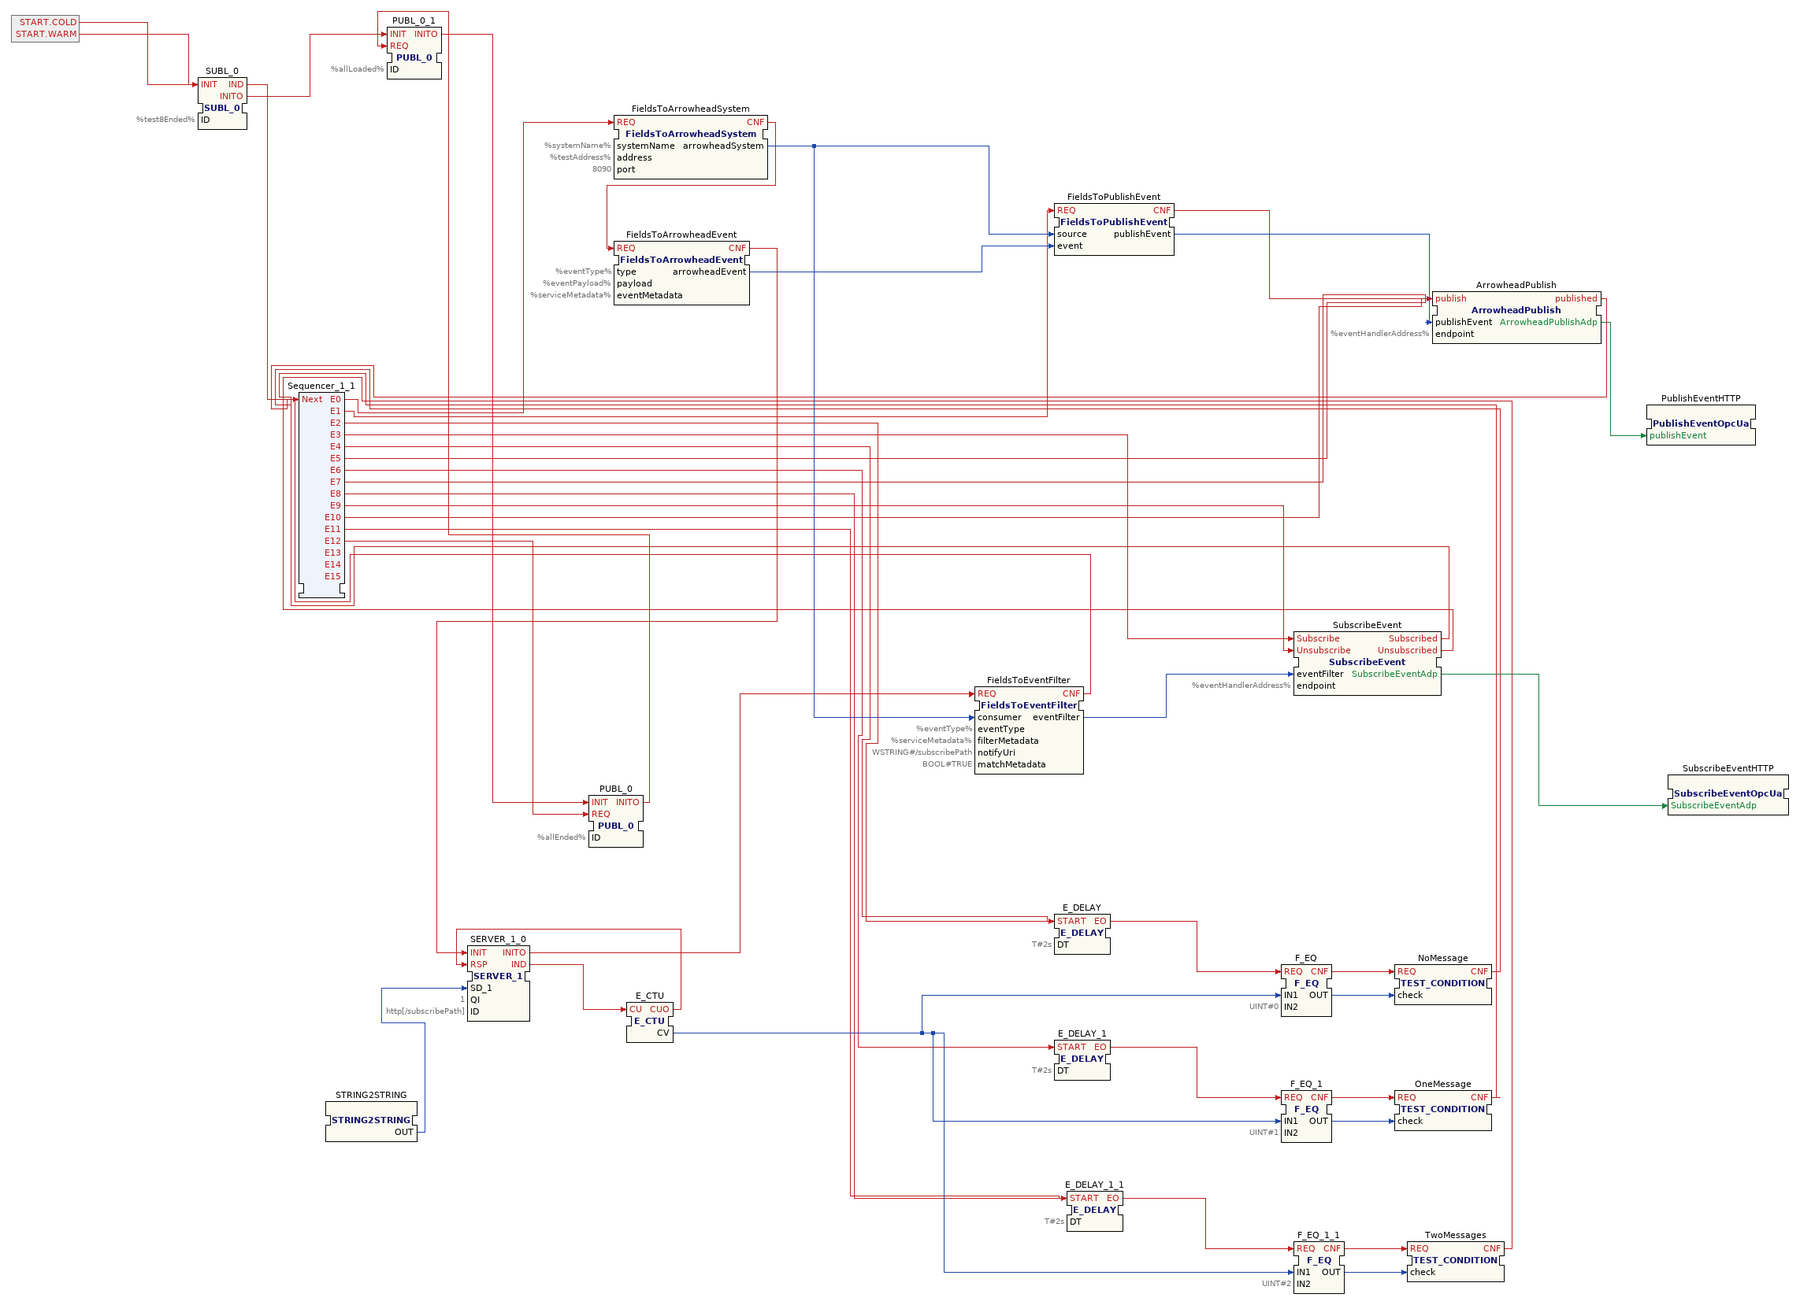
      FBS
        FieldsToPublishEvent : FieldsToPublishEvent;
        FieldsToArrowheadSystem : FieldsToArrowheadSystem(systemName := %systemName%, address := %testAddress%, port := 8090);
        ArrowheadPublish : ArrowheadPublish(endpoint := %eventHandlerAddress%);
        PublishEventHTTP : PublishEventOpcUa;
        FieldsToArrowheadEvent : FieldsToArrowheadEvent(type := %eventType%, payload := %eventPayload%, eventMetadata := %serviceMetadata%);
        FieldsToEventFilter : FieldsToEventFilter(eventType := %eventType%, filterMetadata := %serviceMetadata%, notifyUri := WSTRING#/subscribePath, matchMetadata := BOOL#TRUE);
        SubscribeEvent : SubscribeEvent(endpoint := %eventHandlerAddress%);
        SubscribeEventHTTP : SubscribeEventOpcUa;
        E_CTU : E_CTU;
        F_EQ : F_EQ(IN2 := UINT#0);
        E_DELAY : E_DELAY(DT := T#2s);
        NoMessage : TEST_CONDITION;
        F_EQ_1 : F_EQ(IN2 := UINT#1);
        OneMessage : TEST_CONDITION;
        E_DELAY_1 : E_DELAY(DT := T#2s);
        E_DELAY_1_1 : E_DELAY(DT := T#2s);
        F_EQ_1_1 : F_EQ(IN2 := UINT#2);
        TwoMessages : TEST_CONDITION;
        SUBL_0 : SUBL_0(ID := %test8Ended%);
        PUBL_0_1 : PUBL_0(ID := %allLoaded%);
        PUBL_0 : PUBL_0(ID := %allEnded%);
        SERVER_1_0 : SERVER_1(QI := 1, ID := http[/subscribePath]);
        STRING2STRING : STRING2STRING;
      END_FBS
      SUBAPPLICATION Sequencer_1_1
        EVENT_INPUT
          Next;
        END_EVENT
        EVENT_OUTPUT
          E0;
          E1;
          E2;
          E3;
          E4;
          E5;
          E6;
          E7;
          E8;
          E9;
          E10;
          E11;
          E12;
          E13;
          E14;
          E15;
        END_EVENT
      END_SUBAPPLICATION
      EVENT_CONNECTIONS
        FieldsToPublishEvent.CNF TO ArrowheadPublish.publish;
        FieldsToArrowheadSystem.CNF TO FieldsToArrowheadEvent.REQ;
        E_DELAY.EO TO F_EQ.REQ;
        F_EQ.CNF TO NoMessage.REQ;
        F_EQ_1.CNF TO OneMessage.REQ;
        E_DELAY_1.EO TO F_EQ_1.REQ;
        E_DELAY_1_1.EO TO F_EQ_1_1.REQ;
        F_EQ_1_1.CNF TO TwoMessages.REQ;
        TwoMessages.CNF TO Sequencer_1_1.Next;
        OneMessage.CNF TO Sequencer_1_1.Next;
        NoMessage.CNF TO Sequencer_1_1.Next;
        FieldsToEventFilter.CNF TO Sequencer_1_1.Next;
        ArrowheadPublish.published TO Sequencer_1_1.Next;
        SubscribeEvent.Subscribed TO Sequencer_1_1.Next;
        SubscribeEvent.Unsubscribed TO Sequencer_1_1.Next;
        Sequencer_1_1.E0 TO FieldsToArrowheadSystem.REQ;
        Sequencer_1_1.E1 TO FieldsToPublishEvent.REQ;
        Sequencer_1_1.E2 TO E_DELAY.START;
        Sequencer_1_1.E3 TO SubscribeEvent.Subscribe;
        Sequencer_1_1.E4 TO E_DELAY.START;
        Sequencer_1_1.E5 TO ArrowheadPublish.publish;
        Sequencer_1_1.E6 TO E_DELAY_1.START;
        Sequencer_1_1.E7 TO ArrowheadPublish.publish;
        Sequencer_1_1.E8 TO E_DELAY_1_1.START;
        Sequencer_1_1.E9 TO SubscribeEvent.Unsubscribe;
        Sequencer_1_1.E10 TO ArrowheadPublish.publish;
        Sequencer_1_1.E11 TO E_DELAY_1_1.START;
        SUBL_0.IND TO Sequencer_1_1.Next;
        SUBL_0.INITO TO PUBL_0_1.INIT;
        START.COLD TO SUBL_0.INIT;
        START.WARM TO SUBL_0.INIT;
        PUBL_0_1.INITO TO PUBL_0.INIT;
        Sequencer_1_1.E12 TO PUBL_0.REQ;
        PUBL_0.INITO TO PUBL_0_1.REQ;
        FieldsToArrowheadEvent.CNF TO SERVER_1_0.INIT;
        E_CTU.CUO TO SERVER_1_0.RSP;
        SERVER_1_0.INITO TO FieldsToEventFilter.REQ;
        SERVER_1_0.IND TO E_CTU.CU;
      END_CONNECTIONS
      DATA_CONNECTIONS
        FieldsToArrowheadSystem.arrowheadSystem TO FieldsToPublishEvent.source;
        FieldsToPublishEvent.publishEvent TO ArrowheadPublish.publishEvent;
        FieldsToArrowheadEvent.arrowheadEvent TO FieldsToPublishEvent.event;
        FieldsToArrowheadSystem.arrowheadSystem TO FieldsToEventFilter.consumer;
        FieldsToEventFilter.eventFilter TO SubscribeEvent.eventFilter;
        E_CTU.CV TO F_EQ.IN1;
        F_EQ.OUT TO NoMessage.check;
        E_CTU.CV TO F_EQ_1.IN1;
        F_EQ_1.OUT TO OneMessage.check;
        E_CTU.CV TO F_EQ_1_1.IN1;
        F_EQ_1_1.OUT TO TwoMessages.check;
        STRING2STRING.OUT TO SERVER_1_0.SD_1;
      END_CONNECTIONS
      ADAPTER_CONNECTIONS
        ArrowheadPublish.ArrowheadPublishAdp TO PublishEventHTTP.publishEvent;
        SubscribeEvent.SubscribeEventAdp TO SubscribeEventHTTP.SubscribeEventAdp;
      END_CONNECTIONS
    END_RESOURCE
  END_DEVICE
  MAPPINGS
    HTTPTest1RegisterUnregister.GET_AT_INDEX ON HTTPTest.RegisterUnregister.GET_AT_INDEX;
    HTTPTest1RegisterUnregister.ServiceNotRegisteredPos1 ON HTTPTest.RegisterUnregister.ServiceNotRegisteredPos1;
    HTTPTest1RegisterUnregister.FieldsToServiceQueryForm ON HTTPTest.RegisterUnregister.FieldsToServiceQueryForm;
    HTTPTest1RegisterUnregister.QueryServiceHTTP ON HTTPTest.RegisterUnregister.QueryServiceHTTP;
    HTTPTest1RegisterUnregister.FieldsToArrowheadService ON HTTPTest.RegisterUnregister.FieldsToArrowheadService;
    HTTPTest1RegisterUnregister.F_EQ ON HTTPTest.RegisterUnregister.F_EQ;
    HTTPTest1RegisterUnregister.GetEndpointFromServiceRegistryEntry ON HTTPTest.RegisterUnregister.GetEndpointFromServiceRegistryEntry;
    HTTPTest1RegisterUnregister.QueryService ON HTTPTest.RegisterUnregister.QueryService;
    HTTPTest1RegisterUnregister.Registered ON HTTPTest.RegisterUnregister.Registered;
    HTTPTest1RegisterUnregister.E_SWITCH ON HTTPTest.RegisterUnregister.E_SWITCH;
    HTTPTest1RegisterUnregister.F_EQ_1 ON HTTPTest.RegisterUnregister.F_EQ_1;
    HTTPTest1RegisterUnregister.ServiceRegisteredPos0 ON HTTPTest.RegisterUnregister.ServiceRegisteredPos0;
    HTTPTest1RegisterUnregister.Sequencer ON HTTPTest.RegisterUnregister.Sequencer;
    HTTPTest1RegisterUnregister.RegisterServiceHTTP ON HTTPTest.RegisterUnregister.RegisterServiceHTTP;
    HTTPTest1RegisterUnregister.RegisterService ON HTTPTest.RegisterUnregister.RegisterService;
    HTTPTest1RegisterUnregister.FieldsToServiceRegistryEntry ON HTTPTest.RegisterUnregister.FieldsToServiceRegistryEntry;
    HTTPTest1RegisterUnregister.FieldsToArrowheadSystem ON HTTPTest.RegisterUnregister.FieldsToArrowheadSystem;
    HTTPTest2DoubleRegister.QueryService ON HTTPTest.DoubleRegister.QueryService;
    HTTPTest2DoubleRegister.QueryServiceHTTP ON HTTPTest.DoubleRegister.QueryServiceHTTP;
    HTTPTest2DoubleRegister.GET_AT_INDEX ON HTTPTest.DoubleRegister.GET_AT_INDEX;
    HTTPTest2DoubleRegister.F_EQ ON HTTPTest.DoubleRegister.F_EQ;
    HTTPTest2DoubleRegister.ServiceNotRegisteredPos1 ON HTTPTest.DoubleRegister.ServiceNotRegisteredPos1;
    HTTPTest2DoubleRegister.GetEndpointFromServiceRegistryEntry ON HTTPTest.DoubleRegister.GetEndpointFromServiceRegistryEntry;
    HTTPTest2DoubleRegister.FieldsToArrowheadService ON HTTPTest.DoubleRegister.FieldsToArrowheadService;
    HTTPTest2DoubleRegister.FieldsToServiceQueryForm ON HTTPTest.DoubleRegister.FieldsToServiceQueryForm;
    HTTPTest2DoubleRegister.Registered ON HTTPTest.DoubleRegister.Registered;
    HTTPTest2DoubleRegister.E_SWITCH ON HTTPTest.DoubleRegister.E_SWITCH;
    HTTPTest2DoubleRegister.F_EQ_1 ON HTTPTest.DoubleRegister.F_EQ_1;
    HTTPTest2DoubleRegister.ServiceRegisteredPos0 ON HTTPTest.DoubleRegister.ServiceRegisteredPos0;
    HTTPTest2DoubleRegister.Sequencer ON HTTPTest.DoubleRegister.Sequencer;
    HTTPTest2DoubleRegister.FieldsToArrowheadSystem ON HTTPTest.DoubleRegister.FieldsToArrowheadSystem;
    HTTPTest2DoubleRegister.FieldsToServiceRegistryEntry ON HTTPTest.DoubleRegister.FieldsToServiceRegistryEntry;
    HTTPTest2DoubleRegister.RegisterService ON HTTPTest.DoubleRegister.RegisterService;
    HTTPTest2DoubleRegister.RegisterServiceHTTP ON HTTPTest.DoubleRegister.RegisterServiceHTTP;
    HTTPTest2DoubleRegister.GET_AT_INDEX_1 ON HTTPTest.DoubleRegister.GET_AT_INDEX_1;
    HTTPTest2DoubleRegister.F_EQ_2 ON HTTPTest.DoubleRegister.F_EQ_2;
    HTTPTest2DoubleRegister.ServiceNotRegisteredPos0 ON HTTPTest.DoubleRegister.ServiceNotRegisteredPos0;
    HTTPTest1RegisterUnregister.GetEndpointFromServiceRegistryEntry_1 ON HTTPTest.RegisterUnregister.GetEndpointFromServiceRegistryEntry_1;
    HTTPTest1RegisterUnregister.F_EQ_2 ON HTTPTest.RegisterUnregister.F_EQ_2;
    HTTPTest1RegisterUnregister.ServiceNotRegisteredPos0 ON HTTPTest.RegisterUnregister.ServiceNotRegisteredPos0;
    HTTPTest1RegisterUnregister.GET_AT_INDEX_1 ON HTTPTest.RegisterUnregister.GET_AT_INDEX_1;
    HTTPTest1RegisterUnregister.PUBLISH_0 ON HTTPTest.RegisterUnregister.PUBLISH_0;
    HTTPTest2DoubleRegister.SUBSCRIBE_0 ON HTTPTest.DoubleRegister.SUBSCRIBE_0;
    HTTPTest3RegisterMoreServices.E_SWITCH ON HTTPTest.RegisterMoreServices.E_SWITCH;
    HTTPTest3RegisterMoreServices.GetEndpointFromServiceRegistryEntry_1 ON HTTPTest.RegisterMoreServices.GetEndpointFromServiceRegistryEntry_1;
    HTTPTest3RegisterMoreServices.FieldsToArrowheadSystem ON HTTPTest.RegisterMoreServices.FieldsToArrowheadSystem;
    HTTPTest3RegisterMoreServices.Service2RegisteredPos0 ON HTTPTest.RegisterMoreServices.Service2RegisteredPos0;
    HTTPTest3RegisterMoreServices.Service1RegisteredPos0 ON HTTPTest.RegisterMoreServices.Service1RegisteredPos0;
    HTTPTest3RegisterMoreServices.F_EQ ON HTTPTest.RegisterMoreServices.F_EQ;
    HTTPTest3RegisterMoreServices.F_EQ_2 ON HTTPTest.RegisterMoreServices.F_EQ_2;
    HTTPTest3RegisterMoreServices.GetEndpointFromServiceRegistryEntry ON HTTPTest.RegisterMoreServices.GetEndpointFromServiceRegistryEntry;
    HTTPTest3RegisterMoreServices.Service1NotRegisteredPos1 ON HTTPTest.RegisterMoreServices.Service1NotRegisteredPos1;
    HTTPTest3RegisterMoreServices.Sequencer ON HTTPTest.RegisterMoreServices.Sequencer;
    HTTPTest3RegisterMoreServices.GET_AT_INDEX ON HTTPTest.RegisterMoreServices.GET_AT_INDEX;
    HTTPTest3RegisterMoreServices.GET_AT_INDEX_1 ON HTTPTest.RegisterMoreServices.GET_AT_INDEX_1;
    HTTPTest3RegisterMoreServices.F_EQ_1 ON HTTPTest.RegisterMoreServices.F_EQ_1;
    HTTPTest3RegisterMoreServices.S1Reg ON HTTPTest.RegisterMoreServices.S1Reg;
    HTTPTest3RegisterMoreServices.RegisterService2 ON HTTPTest.RegisterMoreServices.RegisterService2;
    HTTPTest3RegisterMoreServices.RegisterService1 ON HTTPTest.RegisterMoreServices.RegisterService1;
    HTTPTest3RegisterMoreServices.Service2NotRegisteredPos1 ON HTTPTest.RegisterMoreServices.Service2NotRegisteredPos1;
    HTTPTest3RegisterMoreServices.F_EQ_1_1 ON HTTPTest.RegisterMoreServices.F_EQ_1_1;
    HTTPTest3RegisterMoreServices.S2Reg ON HTTPTest.RegisterMoreServices.S2Reg;
    HTTPTest3RegisterMoreServices.E_SWITCH_1 ON HTTPTest.RegisterMoreServices.E_SWITCH_1;
    HTTPTest3RegisterMoreServices.GetEndpointFromServiceRegistryEntry_1_1 ON HTTPTest.RegisterMoreServices.GetEndpointFromServiceRegistryEntry_1_1;
    HTTPTest3RegisterMoreServices.GetEndpointFromServiceRegistryEntry_2 ON HTTPTest.RegisterMoreServices.GetEndpointFromServiceRegistryEntry_2;
    HTTPTest3RegisterMoreServices.GET_AT_INDEX_1_1 ON HTTPTest.RegisterMoreServices.GET_AT_INDEX_1_1;
    HTTPTest3RegisterMoreServices.QueryService2 ON HTTPTest.RegisterMoreServices.QueryService2;
    HTTPTest3RegisterMoreServices.GET_AT_INDEX_2 ON HTTPTest.RegisterMoreServices.GET_AT_INDEX_2;
    HTTPTest3RegisterMoreServices.SUBL_0 ON HTTPTest.RegisterMoreServices.SUBL_0;
    HTTPTest2DoubleRegister.PUBL_0 ON HTTPTest.DoubleRegister.PUBL_0;
    HTTPTest3RegisterMoreServices.F_EQ_3 ON HTTPTest.RegisterMoreServices.F_EQ_3;
    HTTPTest3RegisterMoreServices.Service1NotRegisteredPos0 ON HTTPTest.RegisterMoreServices.Service1NotRegisteredPos0;
    HTTPTest3RegisterMoreServices.F_EQ_3_1 ON HTTPTest.RegisterMoreServices.F_EQ_3_1;
    HTTPTest3RegisterMoreServices.Service2NotRegisteredPos0 ON HTTPTest.RegisterMoreServices.Service2NotRegisteredPos0;
    HTTPTest3RegisterMoreServices.QueryService1 ON HTTPTest.RegisterMoreServices.QueryService1;
    HTTPTest0CleanALL.RegisterService1 ON HTTPTest.cleanAll.RegisterService1;
    HTTPTest0CleanALL.RegisterService2 ON HTTPTest.cleanAll.RegisterService2;
    HTTPTest0CleanALL.FieldsToArrowheadSystem ON HTTPTest.cleanAll.FieldsToArrowheadSystem;
    HTTPTest1RegisterUnregister.SUBL_0 ON HTTPTest.RegisterUnregister.SUBL_0;
    HTTPTest0CleanALL.PUBL_0 ON HTTPTest.cleanAll.PUBL_0;
    HTTPTest0CleanALL.FieldsToArrowheadService ON HTTPTest.cleanAll.FieldsToArrowheadService;
    HTTPTest0CleanALL.FieldsToArrowheadService_1 ON HTTPTest.cleanAll.FieldsToArrowheadService_1;
    HTTPTest3RegisterMoreServices.Service1 ON HTTPTest.RegisterMoreServices.Service1;
    HTTPTest3RegisterMoreServices.Service2 ON HTTPTest.RegisterMoreServices.Service2;
    HTTPTest3RegisterMoreServices.PUBL_0 ON HTTPTest.RegisterMoreServices.PUBL_0;
    HTTPTest4SameServiceTwice.SUBL_0 ON HTTPTest.SameServiceTwice.SUBL_0;
    HTTPTest4SameServiceTwice.Sequencer ON HTTPTest.SameServiceTwice.Sequencer;
    HTTPTest4SameServiceTwice.RegisterService2 ON HTTPTest.SameServiceTwice.RegisterService2;
    HTTPTest4SameServiceTwice.Service1 ON HTTPTest.SameServiceTwice.Service1;
    HTTPTest4SameServiceTwice.RegisterService1 ON HTTPTest.SameServiceTwice.RegisterService1;
    HTTPTest4SameServiceTwice.FieldsToArrowheadSystem ON HTTPTest.SameServiceTwice.FieldsToArrowheadSystem;
    HTTPTest4SameServiceTwice.QueryServiceHTTPSub ON HTTPTest.SameServiceTwice.QueryServiceHTTPSub;
    HTTPTest4SameServiceTwice.GET_AT_INDEX_1 ON HTTPTest.SameServiceTwice.GET_AT_INDEX_1;
    HTTPTest4SameServiceTwice.GetEndpointFromServiceRegistryEntry ON HTTPTest.SameServiceTwice.GetEndpointFromServiceRegistryEntry;
    HTTPTest4SameServiceTwice.GET_AT_INDEX ON HTTPTest.SameServiceTwice.GET_AT_INDEX;
    HTTPTest4SameServiceTwice.GetEndpointFromServiceRegistryEntry_1 ON HTTPTest.SameServiceTwice.GetEndpointFromServiceRegistryEntry_1;
    HTTPTest4SameServiceTwice.Service1RegisteredPos0 ON HTTPTest.SameServiceTwice.Service1RegisteredPos0;
    HTTPTest4SameServiceTwice.F_EQ_2 ON HTTPTest.SameServiceTwice.F_EQ_2;
    HTTPTest4SameServiceTwice.BothServicesRegistered ON HTTPTest.SameServiceTwice.BothServicesRegistered;
    HTTPTest4SameServiceTwice.F_EQ_3 ON HTTPTest.SameServiceTwice.F_EQ_3;
    HTTPTest4SameServiceTwice.F_EQ ON HTTPTest.SameServiceTwice.F_EQ;
    HTTPTest4SameServiceTwice.F_EQ_2_1 ON HTTPTest.SameServiceTwice.F_EQ_2_1;
    HTTPTest4SameServiceTwice.F_EQ_3_1 ON HTTPTest.SameServiceTwice.F_EQ_3_1;
    HTTPTest4SameServiceTwice.Service2RegisteredPos0 ON HTTPTest.SameServiceTwice.Service2RegisteredPos0;
    HTTPTest4SameServiceTwice.F_EQ_1 ON HTTPTest.SameServiceTwice.F_EQ_1;
    HTTPTest4SameServiceTwice.BothServicesNotRegistered ON HTTPTest.SameServiceTwice.BothServicesNotRegistered;
    HTTPTest4SameServiceTwice.F_EQ_1_1 ON HTTPTest.SameServiceTwice.F_EQ_1_1;
    HTTPTest4SameServiceTwice.F_EQ_1_1_1 ON HTTPTest.SameServiceTwice.F_EQ_1_1_1;
    HTTPTest4SameServiceTwice.Service2NotRegisteredPos1 ON HTTPTest.SameServiceTwice.Service2NotRegisteredPos1;
    HTTPTest4SameServiceTwice.F_EQ_4 ON HTTPTest.SameServiceTwice.F_EQ_4;
    HTTPTest4SameServiceTwice.F_EQ_4_1 ON HTTPTest.SameServiceTwice.F_EQ_4_1;
    HTTPTest4SameServiceTwice.Service1NotRegisteredPos1 ON HTTPTest.SameServiceTwice.Service1NotRegisteredPos1;
    HTTPTest4SameServiceTwice.F_AND ON HTTPTest.SameServiceTwice.F_AND;
    HTTPTest4SameServiceTwice.E_MERGE ON HTTPTest.SameServiceTwice.E_MERGE;
    HTTPTest4SameServiceTwice.E_MERGE_1 ON HTTPTest.SameServiceTwice.E_MERGE_1;
    HTTPTest4SameServiceTwice.F_AND_1 ON HTTPTest.SameServiceTwice.F_AND_1;
    HTTPTest4SameServiceTwice.F_OR ON HTTPTest.SameServiceTwice.F_OR;
    HTTPTest4SameServiceTwice.F_AND_1_1 ON HTTPTest.SameServiceTwice.F_AND_1_1;
    HTTPTest4SameServiceTwice.BOOL2BOOL ON HTTPTest.SameServiceTwice.BOOL2BOOL;
    HTTPTest4SameServiceTwice.BOOL2BOOL_1 ON HTTPTest.SameServiceTwice.BOOL2BOOL_1;
    HTTPTest0CleanALL.RegisterService2_1 ON HTTPTest.cleanAll.RegisterService2_1;
    HTTPTest4SameServiceTwice.FieldsToArrowheadSystem_1 ON HTTPTest.SameServiceTwice.FieldsToArrowheadSystem_1;
    HTTPTest0CleanALL.FieldsToArrowheadSystem_1 ON HTTPTest.cleanAll.FieldsToArrowheadSystem_1;
    HTTPTest4SameServiceTwice.PUBL_0 ON HTTPTest.SameServiceTwice.PUBL_0;
    HTTPTest5VersionAndMetadata.RegisterServiceFullHTTP ON HTTPTest.VersionInterfaceAndMetadata.RegisterServiceFullHTTP;
    HTTPTest5VersionAndMetadata.QueryServiceHTTPSub ON HTTPTest.VersionInterfaceAndMetadata.QueryServiceHTTPSub;
    HTTPTest5VersionAndMetadata.FieldsToArrowheadService ON HTTPTest.VersionInterfaceAndMetadata.FieldsToArrowheadService;
    HTTPTest5VersionAndMetadata.GetEndpointFromServiceRegistryEntry ON HTTPTest.VersionInterfaceAndMetadata.GetEndpointFromServiceRegistryEntry;
    HTTPTest5VersionAndMetadata.GET_AT_INDEX ON HTTPTest.VersionInterfaceAndMetadata.GET_AT_INDEX;
    HTTPTest5VersionAndMetadata.F_EQ_4 ON HTTPTest.VersionInterfaceAndMetadata.F_EQ_4;
    HTTPTest5VersionAndMetadata.LowerVersion ON HTTPTest.VersionInterfaceAndMetadata.LowerVersion;
    HTTPTest5VersionAndMetadata.FieldsToArrowheadService_1 ON HTTPTest.VersionInterfaceAndMetadata.FieldsToArrowheadService_1;
    HTTPTest5VersionAndMetadata.SameVersion ON HTTPTest.VersionInterfaceAndMetadata.SameVersion;
    HTTPTest5VersionAndMetadata.QueryServiceHTTPSub_1 ON HTTPTest.VersionInterfaceAndMetadata.QueryServiceHTTPSub_1;
    HTTPTest5VersionAndMetadata.GET_AT_INDEX_1 ON HTTPTest.VersionInterfaceAndMetadata.GET_AT_INDEX_1;
    HTTPTest5VersionAndMetadata.GetEndpointFromServiceRegistryEntry_1 ON HTTPTest.VersionInterfaceAndMetadata.GetEndpointFromServiceRegistryEntry_1;
    HTTPTest5VersionAndMetadata.F_EQ_4_1 ON HTTPTest.VersionInterfaceAndMetadata.F_EQ_4_1;
    HTTPTest5VersionAndMetadata.OneInterfaceOutOfTwo ON HTTPTest.VersionInterfaceAndMetadata.OneInterfaceOutOfTwo;
    HTTPTest5VersionAndMetadata.QueryServiceHTTPSub_1_1 ON HTTPTest.VersionInterfaceAndMetadata.QueryServiceHTTPSub_1_1;
    HTTPTest5VersionAndMetadata.GetEndpointFromServiceRegistryEntry_1_1 ON HTTPTest.VersionInterfaceAndMetadata.GetEndpointFromServiceRegistryEntry_1_1;
    HTTPTest5VersionAndMetadata.F_EQ_4_1_1 ON HTTPTest.VersionInterfaceAndMetadata.F_EQ_4_1_1;
    HTTPTest5VersionAndMetadata.FieldsToArrowheadService_1_1 ON HTTPTest.VersionInterfaceAndMetadata.FieldsToArrowheadService_1_1;
    HTTPTest5VersionAndMetadata.GET_AT_INDEX_1_1 ON HTTPTest.VersionInterfaceAndMetadata.GET_AT_INDEX_1_1;
    HTTPTest5VersionAndMetadata.OneInterfaceOutOfTwo_2 ON HTTPTest.VersionInterfaceAndMetadata.OneInterfaceOutOfTwo_2;
    HTTPTest5VersionAndMetadata.QueryServiceHTTPSub_1_2 ON HTTPTest.VersionInterfaceAndMetadata.QueryServiceHTTPSub_1_2;
    HTTPTest5VersionAndMetadata.GetEndpointFromServiceRegistryEntry_1_2 ON HTTPTest.VersionInterfaceAndMetadata.GetEndpointFromServiceRegistryEntry_1_2;
    HTTPTest5VersionAndMetadata.F_EQ_4_1_2 ON HTTPTest.VersionInterfaceAndMetadata.F_EQ_4_1_2;
    HTTPTest5VersionAndMetadata.FieldsToArrowheadService_1_2 ON HTTPTest.VersionInterfaceAndMetadata.FieldsToArrowheadService_1_2;
    HTTPTest5VersionAndMetadata.GET_AT_INDEX_1_2 ON HTTPTest.VersionInterfaceAndMetadata.GET_AT_INDEX_1_2;
    HTTPTest5VersionAndMetadata.WrongInterface ON HTTPTest.VersionInterfaceAndMetadata.WrongInterfaceProvided;
    HTTPTest5VersionAndMetadata.GET_AT_INDEX_1_2_1 ON HTTPTest.VersionInterfaceAndMetadata.GET_AT_INDEX_1_2_1;
    HTTPTest5VersionAndMetadata.QueryServiceHTTPSub_1_2_1 ON HTTPTest.VersionInterfaceAndMetadata.QueryServiceHTTPSub_1_2_1;
    HTTPTest5VersionAndMetadata.GetEndpointFromServiceRegistryEntry_1_2_1 ON HTTPTest.VersionInterfaceAndMetadata.GetEndpointFromServiceRegistryEntry_1_2_1;
    HTTPTest5VersionAndMetadata.FieldsToArrowheadService_1_2_1 ON HTTPTest.VersionInterfaceAndMetadata.FieldsToArrowheadService_1_2_1;
    HTTPTest5VersionAndMetadata.F_EQ_4_1_2_1 ON HTTPTest.VersionInterfaceAndMetadata.F_EQ_4_1_2_1;
    HTTPTest5VersionAndMetadata.SUBL_0 ON HTTPTest.VersionInterfaceAndMetadata.SUBL_0;
    HTTPTest5VersionAndMetadata.OnlyOneMetadata ON HTTPTest.VersionInterfaceAndMetadata.OnlyOneMetadata;
    HTTPTest5VersionAndMetadata.GetEndpointFromServiceRegistryEntry_1_2_1_1 ON HTTPTest.VersionInterfaceAndMetadata.GetEndpointFromServiceRegistryEntry_1_2_1_1;
    HTTPTest5VersionAndMetadata.F_EQ_4_1_2_1_1 ON HTTPTest.VersionInterfaceAndMetadata.F_EQ_4_1_2_1_1;
    HTTPTest5VersionAndMetadata.FieldsToArrowheadService_1_2_1_1 ON HTTPTest.VersionInterfaceAndMetadata.FieldsToArrowheadService_1_2_1_1;
    HTTPTest5VersionAndMetadata.GET_AT_INDEX_1_2_1_1 ON HTTPTest.VersionInterfaceAndMetadata.GET_AT_INDEX_1_2_1_1;
    HTTPTest5VersionAndMetadata.QueryServiceHTTPSub_1_2_1_1 ON HTTPTest.VersionInterfaceAndMetadata.QueryServiceHTTPSub_1_2_1_1;
    HTTPTest5VersionAndMetadata.QueryServiceHTTPSub_1_2_1_1_1 ON HTTPTest.VersionInterfaceAndMetadata.QueryServiceHTTPSub_1_2_1_1_1;
    HTTPTest5VersionAndMetadata.GetEndpointFromServiceRegistryEntry_1_2_1_1_1 ON HTTPTest.VersionInterfaceAndMetadata.GetEndpointFromServiceRegistryEntry_1_2_1_1_1;
    HTTPTest5VersionAndMetadata.FieldsToArrowheadService_1_2_1_1_1 ON HTTPTest.VersionInterfaceAndMetadata.FieldsToArrowheadService_1_2_1_1_1;
    HTTPTest5VersionAndMetadata.F_EQ_4_1_2_1_1_1 ON HTTPTest.VersionInterfaceAndMetadata.F_EQ_4_1_2_1_1_1;
    HTTPTest5VersionAndMetadata.GET_AT_INDEX_1_2_1_1_1 ON HTTPTest.VersionInterfaceAndMetadata.GET_AT_INDEX_1_2_1_1_1;
    HTTPTest5VersionAndMetadata.NoMetadataAndAsked ON HTTPTest.VersionInterfaceAndMetadata.NoMetadataAndAsked;
    HTTPTest5VersionAndMetadata.FieldsToArrowheadService_1_2_1_2 ON HTTPTest.VersionInterfaceAndMetadata.FieldsToArrowheadService_1_2_1_2;
    HTTPTest5VersionAndMetadata.F_EQ_4_1_2_1_2 ON HTTPTest.VersionInterfaceAndMetadata.F_EQ_4_1_2_1_2;
    HTTPTest5VersionAndMetadata.GetEndpointFromServiceRegistryEntry_1_2_1_2 ON HTTPTest.VersionInterfaceAndMetadata.GetEndpointFromServiceRegistryEntry_1_2_1_2;
    HTTPTest5VersionAndMetadata.GET_AT_INDEX_1_2_1_2 ON HTTPTest.VersionInterfaceAndMetadata.GET_AT_INDEX_1_2_1_2;
    HTTPTest5VersionAndMetadata.NoInterface ON HTTPTest.VersionInterfaceAndMetadata.NoInterfaceProvided;
    HTTPTest5VersionAndMetadata.QueryServiceHTTPSub_1_2_1_2 ON HTTPTest.VersionInterfaceAndMetadata.QueryServiceHTTPSub_1_2_1_2;
    HTTPTest5VersionAndMetadata.GET_AT_INDEX_1_2_1_1_1_1 ON HTTPTest.VersionInterfaceAndMetadata.GET_AT_INDEX_1_2_1_1_1_1;
    HTTPTest5VersionAndMetadata.FieldsToArrowheadService_1_2_1_1_1_1 ON HTTPTest.VersionInterfaceAndMetadata.FieldsToArrowheadService_1_2_1_1_1_1;
    HTTPTest5VersionAndMetadata.WrongMetadaButNotAsked ON HTTPTest.VersionInterfaceAndMetadata.WrongMetadaButNotAsked;
    HTTPTest5VersionAndMetadata.QueryServiceHTTPSub_1_2_1_1_1_1 ON HTTPTest.VersionInterfaceAndMetadata.QueryServiceHTTPSub_1_2_1_1_1_1;
    HTTPTest5VersionAndMetadata.GetEndpointFromServiceRegistryEntry_1_2_1_1_1_1 ON HTTPTest.VersionInterfaceAndMetadata.GetEndpointFromServiceRegistryEntry_1_2_1_1_1_1;
    HTTPTest5VersionAndMetadata.F_EQ_4_1_2_1_1_1_1 ON HTTPTest.VersionInterfaceAndMetadata.F_EQ_4_1_2_1_1_1_1;
    HTTPTest0CleanALL.SUBL_0 ON HTTPTest.cleanAll.SUBL_0;
    HTTPTest0CleanALL.STEST_END ON HTTPTest.cleanAll.STEST_END;
    HTTPTest5VersionAndMetadata.PUBL_0 ON HTTPTest.VersionInterfaceAndMetadata.PUBL_0;
    HTTPTest6RegisterMoreServiceSubApp.SUBL_0 ON HTTPTest.RegisterMoreServicesSubApp.SUBL_0;
    HTTPTest6RegisterMoreServiceSubApp.GetEndpointFromServiceRegistryEntry_1 ON HTTPTest.RegisterMoreServicesSubApp.GetEndpointFromServiceRegistryEntry_1;
    HTTPTest6RegisterMoreServiceSubApp.GET_AT_INDEX_1 ON HTTPTest.RegisterMoreServicesSubApp.GET_AT_INDEX_1;
    HTTPTest6RegisterMoreServiceSubApp.GetEndpointFromServiceRegistryEntry ON HTTPTest.RegisterMoreServicesSubApp.GetEndpointFromServiceRegistryEntry;
    HTTPTest6RegisterMoreServiceSubApp.FieldsToArrowheadSystem ON HTTPTest.RegisterMoreServicesSubApp.FieldsToArrowheadSystem;
    HTTPTest6RegisterMoreServiceSubApp.F_EQ_2 ON HTTPTest.RegisterMoreServicesSubApp.F_EQ_2;
    HTTPTest6RegisterMoreServiceSubApp.GET_AT_INDEX ON HTTPTest.RegisterMoreServicesSubApp.GET_AT_INDEX;
    HTTPTest6RegisterMoreServiceSubApp.Pos1Empty2 ON HTTPTest.RegisterMoreServicesSubApp.Pos1Empty2;
    HTTPTest6RegisterMoreServiceSubApp.F_EQ_1 ON HTTPTest.RegisterMoreServicesSubApp.F_EQ_1;
    HTTPTest6RegisterMoreServiceSubApp.Pos1Empty ON HTTPTest.RegisterMoreServicesSubApp.Pos1Empty;
    HTTPTest6RegisterMoreServiceSubApp.Sequencer ON HTTPTest.RegisterMoreServicesSubApp.Sequencer;
    HTTPTest6RegisterMoreServiceSubApp.GET_AT_INDEX_1_1 ON HTTPTest.RegisterMoreServicesSubApp.GET_AT_INDEX_1_1;
    HTTPTest6RegisterMoreServiceSubApp.GetEndpointFromServiceRegistryEntry_1_1 ON HTTPTest.RegisterMoreServicesSubApp.GetEndpointFromServiceRegistryEntry_1_1;
    HTTPTest6RegisterMoreServiceSubApp.GetEndpointFromServiceRegistryEntry_2 ON HTTPTest.RegisterMoreServicesSubApp.GetEndpointFromServiceRegistryEntry_2;
    HTTPTest6RegisterMoreServiceSubApp.GET_AT_INDEX_2 ON HTTPTest.RegisterMoreServicesSubApp.GET_AT_INDEX_2;
    HTTPTest6RegisterMoreServiceSubApp.Pos0Service1 ON HTTPTest.RegisterMoreServicesSubApp.Pos0Service1;
    HTTPTest6RegisterMoreServiceSubApp.F_EQ_3 ON HTTPTest.RegisterMoreServicesSubApp.F_EQ_3;
    HTTPTest6RegisterMoreServiceSubApp.F_EQ_3_1 ON HTTPTest.RegisterMoreServicesSubApp.F_EQ_3_1;
    HTTPTest6RegisterMoreServiceSubApp.Pos0Service2 ON HTTPTest.RegisterMoreServicesSubApp.Pos0Service2;
    HTTPTest6RegisterMoreServiceSubApp.PUBL_0_1 ON HTTPTest.RegisterMoreServicesSubApp.PUBL_0_1;
    HTTPTest6RegisterMoreServiceSubApp.QuerySecondService ON HTTPTest.RegisterMoreServicesSubApp.QuerySecondService;
    HTTPTest6RegisterMoreServiceSubApp.QueryFirstService ON HTTPTest.RegisterMoreServicesSubApp.QueryFirstService;
    HTTPTest6RegisterMoreServiceSubApp.F_EQ_1_1 ON HTTPTest.RegisterMoreServicesSubApp.F_EQ_1_1;
    HTTPTest6RegisterMoreServiceSubApp.F_EQ_3_1_1 ON HTTPTest.RegisterMoreServicesSubApp.F_EQ_3_1_1;
    HTTPTest6RegisterMoreServiceSubApp.Pos1Empty3 ON HTTPTest.RegisterMoreServicesSubApp.Pos1Empty3;
    HTTPTest6RegisterMoreServiceSubApp.Pos0Empty3 ON HTTPTest.RegisterMoreServicesSubApp.Pos0Empty3;
    HTTPTest6RegisterMoreServiceSubApp.F_EQ_1_1_1 ON HTTPTest.RegisterMoreServicesSubApp.F_EQ_1_1_1;
    HTTPTest6RegisterMoreServiceSubApp.Pos0Empty4 ON HTTPTest.RegisterMoreServicesSubApp.Pos0Empty4;
    HTTPTest6RegisterMoreServiceSubApp.Pos1Empty4 ON HTTPTest.RegisterMoreServicesSubApp.Pos1Empty4;
    HTTPTest6RegisterMoreServiceSubApp.F_EQ_3_1_1_1 ON HTTPTest.RegisterMoreServicesSubApp.F_EQ_3_1_1_1;
    HTTPTest6RegisterMoreServiceSubApp.E_MERGE ON HTTPTest.RegisterMoreServicesSubApp.E_MERGE;
    HTTPTest6RegisterMoreServiceSubApp.E_MERGE_1 ON HTTPTest.RegisterMoreServicesSubApp.E_MERGE_1;
    HTTPTest6RegisterMoreServiceSubApp.RegisterManyServices ON HTTPTest.RegisterMoreServicesSubApp.RegisterManyServices;
    HTTPTest7OrchestrationNoRules.RequestOrchestrationHTTP ON HTTPTest.OrchestratorNoRule.RequestOrchestrationHTTP;
    HTTPTest7OrchestrationNoRules.FieldsToServiceRequestForm ON HTTPTest.OrchestratorNoRule.FieldsToServiceRequestForm;
    HTTPTest7OrchestrationNoRules.FieldsToArrowheadSystem ON HTTPTest.OrchestratorNoRule.FieldsToArrowheadSystem;
    HTTPTest7OrchestrationNoRules.Service1 ON HTTPTest.OrchestratorNoRule.Service1;
    HTTPTest7OrchestrationNoRules.GetEndpointFromOrchestrationForm ON HTTPTest.OrchestratorNoRule.GetEndpointFromOrchestrationForm;
    HTTPTest7OrchestrationNoRules.F_EQ ON HTTPTest.OrchestratorNoRule.F_EQ;
    HTTPTest7OrchestrationNoRules.NoServiceAvailable ON HTTPTest.OrchestratorNoRule.NoServiceAvailable;
    HTTPTest7OrchestrationNoRules.SERVER_1 ON HTTPTest.OrchestratorNoRule.SERVER_1;
    HTTPTest7OrchestrationNoRules.E_SR ON HTTPTest.OrchestratorNoRule.E_SR;
    HTTPTest7OrchestrationNoRules.RegisterService2 ON HTTPTest.OrchestratorNoRule.RegisterService2;
    HTTPTest7OrchestrationNoRules.SUBL_0 ON HTTPTest.OrchestratorNoRule.SUBL_0;
    HTTPTest7OrchestrationNoRules.PUBL_0 ON HTTPTest.OrchestratorNoRule.PUBL_0;
    HTTPTest7OrchestrationNoRules.GET_STRUCT_VALUE1 ON HTTPTest.OrchestratorNoRule.GET_STRUCT_VALUE1;
    HTTPTest7OrchestrationNoRules.Sequencer_1 ON HTTPTest.OrchestratorNoRule.Sequencer_1;
    HTTPTest8OrchestrationWithRules.FieldsToArrowheadSystem ON HTTPTest.OrchestrationWithRules.FieldsToArrowheadSystem;
    HTTPTest8OrchestrationWithRules.Service1 ON HTTPTest.OrchestrationWithRules.Service1;
    HTTPTest8OrchestrationWithRules.F_EQ ON HTTPTest.OrchestrationWithRules.F_EQ;
    HTTPTest8OrchestrationWithRules.NoServiceAvailable ON HTTPTest.OrchestrationWithRules.NoServiceAvailable;
    HTTPTest8OrchestrationWithRules.SERVER_1 ON HTTPTest.OrchestrationWithRules.SERVER_1;
    HTTPTest8OrchestrationWithRules.E_SR ON HTTPTest.OrchestrationWithRules.E_SR;
    HTTPTest8OrchestrationWithRules.RegisterService2 ON HTTPTest.OrchestrationWithRules.RegisterService2;
    HTTPTest8OrchestrationWithRules.SUBL_0 ON HTTPTest.OrchestrationWithRules.SUBL_0;
    HTTPTest8OrchestrationWithRules.PUBL_0 ON HTTPTest.OrchestrationWithRules.PUBL_0;
    HTTPTest8OrchestrationWithRules.Sequencer_1 ON HTTPTest.OrchestrationWithRules.Sequencer_1;
    HTTPTest8OrchestrationWithRules.F_EQ_1 ON HTTPTest.OrchestrationWithRules.F_EQ_1;
    HTTPTest8OrchestrationWithRules.ServiceAvailable ON HTTPTest.OrchestrationWithRules.ServiceAvailable;
    HTTPTest8OrchestrationWithRules.E_SR_1 ON HTTPTest.OrchestrationWithRules.E_SR_1;
    HTTPTest8OrchestrationWithRules.E_SWITCH ON HTTPTest.OrchestrationWithRules.E_SWITCH;
    HTTPTest8OrchestrationWithRules.CLIENT_1_2 ON HTTPTest.OrchestrationWithRules.CLIENT_1_2;
    HTTPTest8OrchestrationWithRules.CLIENT_1_2_1 ON HTTPTest.OrchestrationWithRules.CLIENT_1_2_1;
    HTTPTest8OrchestrationWithRules.STRING2STRING ON HTTPTest.OrchestrationWithRules.STRING2STRING;
    HTTPTest0CleanALL.SUBL_0_1 ON HTTPTest.cleanAll.SUBL_0_1;
    HTTPTest7OrchestrationNoRules.RequestOrchestrationForm ON HTTPTest.OrchestratorNoRule.RequestOrchestrationForm;
    HTTPTest2DoubleRegister.GetEndpointFromServiceRegistryEntry_1 ON HTTPTest.DoubleRegister.GetEndpointFromServiceRegistryEntry_1;
    HTTPTest9PublishSubscribe.FieldsToArrowheadSystem ON HTTPTest.PublishSubscribe.FieldsToArrowheadSystem;
    HTTPTest9PublishSubscribe.FieldsToPublishEvent ON HTTPTest.PublishSubscribe.FieldsToPublishEvent;
    HTTPTest9PublishSubscribe.ArrowheadPublish ON HTTPTest.PublishSubscribe.ArrowheadPublish;
    HTTPTest9PublishSubscribe.FieldsToArrowheadEvent ON HTTPTest.PublishSubscribe.FieldsToArrowheadEvent;
    HTTPTest9PublishSubscribe.SubscribeEvent ON HTTPTest.PublishSubscribe.SubscribeEvent;
    HTTPTest9PublishSubscribe.FieldsToEventFilter ON HTTPTest.PublishSubscribe.FieldsToEventFilter;
    HTTPTest9PublishSubscribe.E_CTU ON HTTPTest.PublishSubscribe.E_CTU;
    HTTPTest9PublishSubscribe.F_EQ ON HTTPTest.PublishSubscribe.F_EQ;
    HTTPTest9PublishSubscribe.E_DELAY ON HTTPTest.PublishSubscribe.E_DELAY;
    HTTPTest9PublishSubscribe.NoMessage ON HTTPTest.PublishSubscribe.NoMessage;
    HTTPTest9PublishSubscribe.E_DELAY_1 ON HTTPTest.PublishSubscribe.E_DELAY_1;
    HTTPTest9PublishSubscribe.F_EQ_1 ON HTTPTest.PublishSubscribe.F_EQ_1;
    HTTPTest9PublishSubscribe.OneMessage ON HTTPTest.PublishSubscribe.OneMessage;
    HTTPTest9PublishSubscribe.E_DELAY_1_1 ON HTTPTest.PublishSubscribe.E_DELAY_1_1;
    HTTPTest9PublishSubscribe.TwoMessages ON HTTPTest.PublishSubscribe.TwoMessages;
    HTTPTest9PublishSubscribe.F_EQ_1_1 ON HTTPTest.PublishSubscribe.F_EQ_1_1;
    HTTPTest9PublishSubscribe.Sequencer_1_1 ON HTTPTest.PublishSubscribe.Sequencer_1_1;
    HTTPTest8OrchestrationWithRules.GetEndpointFromOrchestrationHTTPPFull ON HTTPTest.OrchestrationWithRules.GetEndpointFromOrchestrationHTTPPFull;
    HTTPTest9PublishSubscribe.SERVER_1_0 ON HTTPTest.PublishSubscribe.SERVER_1_0;
    HTTPTest9PublishSubscribe.PUBL_0_1 ON HTTPTest.PublishSubscribe.PUBL_0_1;
    HTTPTest9PublishSubscribe.SUBL_0 ON HTTPTest.PublishSubscribe.SUBL_0;
    HTTPTest9PublishSubscribe.PUBL_0 ON HTTPTest.PublishSubscribe.PUBL_0;
    HTTPTest9PublishSubscribe.PublishEventHTTP ON HTTPTest.PublishSubscribe.PublishEventHTTP;
    HTTPTest9PublishSubscribe.SubscribeEventHTTP ON HTTPTest.PublishSubscribe.SubscribeEventHTTP;
    OpcUaTest0CleanALL.PUBL_0 ON OpcUaTest.cleanAll.PUBL_0;
    OpcUaTest0CleanALL.FieldsToArrowheadSystem ON OpcUaTest.cleanAll.FieldsToArrowheadSystem;
    OpcUaTest0CleanALL.FieldsToArrowheadService ON OpcUaTest.cleanAll.FieldsToArrowheadService;
    OpcUaTest0CleanALL.FieldsToArrowheadService_1 ON OpcUaTest.cleanAll.FieldsToArrowheadService_1;
    OpcUaTest0CleanALL.FieldsToArrowheadSystem_1 ON OpcUaTest.cleanAll.FieldsToArrowheadSystem_1;
    OpcUaTest0CleanALL.SUBL_0 ON OpcUaTest.cleanAll.SUBL_0;
    OpcUaTest0CleanALL.STEST_END ON OpcUaTest.cleanAll.STEST_END;
    OpcUaTest0CleanALL.SUBL_0_1 ON OpcUaTest.cleanAll.SUBL_0_1;
    OpcUaTest1RegisterUnregister.QueryService ON OpcUaTest.RegisterUnregister.QueryService;
    OpcUaTest1RegisterUnregister.GET_AT_INDEX ON OpcUaTest.RegisterUnregister.GET_AT_INDEX;
    OpcUaTest1RegisterUnregister.F_EQ ON OpcUaTest.RegisterUnregister.F_EQ;
    OpcUaTest1RegisterUnregister.ServiceNotRegisteredPos1 ON OpcUaTest.RegisterUnregister.ServiceNotRegisteredPos1;
    OpcUaTest1RegisterUnregister.GetEndpointFromServiceRegistryEntry ON OpcUaTest.RegisterUnregister.GetEndpointFromServiceRegistryEntry;
